LIN {X 0,Y 481.475,Z 710.731,A -85,B 0,C 180,E1 17774.011,E2 17774.011} C_VEL
LIN {X 0,Y 472.315,Z 949.794,A -85,B 0,C 180,E1 17770.464,E2 17770.464} C_VEL
LIN {X 0,Y 470.327,Z 972.285,A -85,B 0,C 180,E1 17769.967,E2 17769.967} C_VEL
LIN {X 0,Y 467.755,Z 993.239,A -85,B 0,C 180,E1 17769.33,E2 17769.33} C_VEL
LIN {X 0,Y 464.62,Z 1013.152,A -85,B 0,C 180,E1 17768.521,E2 17768.521} C_VEL
LIN {X 0,Y 460.838,Z 1033.611,A -85,B 0,C 180,E1 17767.487,E2 17767.487} C_VEL
LIN {X 0,Y 456.775,Z 1052.502,A -85,B 0,C 180,E1 17766.307,E2 17766.307} C_VEL
LIN {X 0,Y 451.974,Z 1072.368,A -85,B 0,C 180,E1 17764.802,E2 17764.802} C_VEL
LIN {X 0,Y 447.338,Z 1090.041,A -85,B 0,C 180,E1 17763.203,E2 17763.203} C_VEL
LIN {X 0,Y 442.542,Z 1106.778,A -85,B 0,C 180,E1 17761.385,E2 17761.385} C_VEL
LIN {X 0,Y 437.61,Z 1123.269,A -85,B 0,C 180,E1 17759.272,E2 17759.272} C_VEL
LIN {X 0,Y 433.368,Z 1137.028,A -85,B 0,C 180,E1 17757.182,E2 17757.182} C_VEL
LIN {X 0,Y 428.992,Z 1151.061,A -85,B 0,C 180,E1 17754.658,E2 17754.658} C_VEL
LIN {X 0,Y 425.363,Z 1163.083,A -85,B 0,C 180,E1 17752.092,E2 17752.092} C_VEL
LIN {X 0,Y 422.273,Z 1173.636,A -85,B 0,C 180,E1 17749.359,E2 17749.359} C_VEL
LIN {X 0,Y 419.714,Z 1183.269,A -85,B 0,C 180,E1 17746.326,E2 17746.326} C_VEL
LIN {X 0,Y 417.954,Z 1191.051,A -85,B 0,C 180,E1 17743.277,E2 17743.277} C_VEL
LIN {X 0,Y 416.861,Z 1196.958,A -85,B 0,C 180,E1 17740.224,E2 17740.224} C_VEL
LIN {X 0,Y 416.258,Z 1201.444,A -85,B 0,C 180,E1 17737.037,E2 17737.037} C_VEL
LIN {X 0,Y 416.044,Z 1204.09,A -85,B 0,C 180,E1 17734.134,E2 17734.134} C_VEL
LIN {X 0,Y 415.975,Z 1205.344,A -85,B 0,C 180,E1 17731.102,E2 17731.102} C_VEL
LIN {X 0,Y 415.981,Z 1205.255,A -85,B 0,C 180,E1 17728.209,E2 17728.209} C_VEL
LIN {X 0,Y 416,Z 1204.756,A -85,B 0,C 180,E1 17726.998,E2 17726.998} C_VEL
LIN {X 0,Y 415.038,Z 1204.26,A -85,B 0,C 180,E1 17725.939,E2 17725.939} C_VEL
LIN {X 0,Y 408.881,Z 1201.972,A -85,B 0,C 180,E1 17723.038,E2 17723.038} C_VEL
LIN {X 0,Y 408.362,Z 1201.086,A -85,B 0,C 180,E1 17722.189,E2 17722.189} C_VEL
LIN {X 0,Y 409.017,Z 1196.625,A -85,B 0,C 180,E1 17719.151,E2 17719.151} C_VEL
LIN {X 0,Y 410.248,Z 1190.54,A -85,B 0,C 180,E1 17716.038,E2 17716.038} C_VEL
LIN {X 0,Y 412.086,Z 1183.005,A -85,B 0,C 180,E1 17713.073,E2 17713.073} C_VEL
LIN {X 0,Y 414.825,Z 1173.243,A -85,B 0,C 180,E1 17709.985,E2 17709.985} C_VEL
LIN {X 0,Y 418.117,Z 1162.59,A -85,B 0,C 180,E1 17707.207,E2 17707.207} C_VEL
LIN {X 0,Y 421.961,Z 1150.464,A -85,B 0,C 180,E1 17704.603,E2 17704.603} C_VEL
LIN {X 0,Y 426.557,Z 1136.278,A -85,B 0,C 180,E1 17702.043,E2 17702.043} C_VEL
LIN {X 0,Y 431.32,Z 1121.527,A -85,B 0,C 180,E1 17699.799,E2 17699.799} C_VEL
LIN {X 0,Y 436.334,Z 1105.207,A -85,B 0,C 180,E1 17697.729,E2 17697.729} C_VEL
LIN {X 0,Y 441.692,Z 1086.828,A -85,B 0,C 180,E1 17695.769,E2 17695.769} C_VEL
LIN {X 0,Y 446.584,Z 1068.818,A -85,B 0,C 180,E1 17694.164,E2 17694.164} C_VEL
LIN {X 0,Y 451.18,Z 1049.908,A -85,B 0,C 180,E1 17692.772,E2 17692.772} C_VEL
LIN {X 0,Y 455.414,Z 1030.616,A -85,B 0,C 180,E1 17691.587,E2 17691.587} C_VEL
LIN {X 0,Y 459.136,Z 1010.497,A -85,B 0,C 180,E1 17690.595,E2 17690.595} C_VEL
LIN {X 0,Y 462.65,Z 987.669,A -85,B 0,C 180,E1 17689.714,E2 17689.714} C_VEL
LIN {X 0,Y 465.3,Z 965.816,A -85,B 0,C 180,E1 17689.089,E2 17689.089} C_VEL
LIN {X 0,Y 466.986,Z 943.197,A -85,B 0,C 180,E1 17688.645,E2 17688.645} C_VEL
LIN {X 0,Y 476.077,Z 710.457,A -85,B 0,C 180,E1 17685.156,E2 17685.156} C_VEL
LIN {X 0,Y 469.155,Z 656.336,A -85,B 0,C 180,E1 17683.01,E2 17683.01} C_VEL
LIN {X 0,Y 466.065,Z 634.46,A -85,B 0,C 180,E1 17682.048,E2 17682.048} C_VEL
LIN {X 0,Y 456.423,Z 617.63,A -85,B 0,C 180,E1 17680.055,E2 17680.055} C_VEL
LIN {X 0,Y 450.65,Z 602.406,A -85,B 0,C 180,E1 17677.122,E2 17677.122} C_VEL
LIN {X 0,Y 445.079,Z 588.882,A -85,B 0,C 180,E1 17674.169,E2 17674.169} C_VEL
LIN {X 0,Y 439.764,Z 577.056,A -85,B 0,C 180,E1 17671.225,E2 17671.225} C_VEL
LIN {X 0,Y 435.667,Z 568.47,A -85,B 0,C 180,E1 17668.814,E2 17668.814} C_VEL
LIN {X 0,Y 431.849,Z 560.755,A -85,B 0,C 180,E1 17666.395,E2 17666.395} C_VEL
LIN {X 0,Y 429.847,Z 556.829,A -85,B 0,C 180,E1 17665.047,E2 17665.047} C_VEL
LIN {X 0,Y 427.57,Z 552.442,A -85,B 0,C 180,E1 17663.425,E2 17663.425} C_VEL
LIN {X 0,Y 425.289,Z 548.024,A -85,B 0,C 180,E1 17661.662,E2 17661.662} C_VEL
LIN {X 0,Y 422.487,Z 542.947,A -85,B 0,C 180,E1 17659.35,E2 17659.35} C_VEL
LIN {X 0,Y 420.43,Z 539.195,A -85,B 0,C 180,E1 17657.437,E2 17657.437} C_VEL
LIN {X 0,Y 419.548,Z 537.819,A -85,B 0,C 180,E1 17656.618,E2 17656.618} C_VEL
LIN {X 0,Y 417.256,Z 533.439,A -85,B 0,C 180,E1 17653.955,E2 17653.955} C_VEL
LIN {X 0,Y 413.712,Z 527.549,A -85,B 0,C 180,E1 17648.758,E2 17648.758} C_VEL
LIN {X 0,Y 411.429,Z 524.761,A -85,B 0,C 180,E1 17643.065,E2 17643.065} C_VEL
LIN {X 0,Y 411.214,Z 524.355,A -85,B 0,C 180,E1 17639.443,E2 17639.443} C_VEL
LIN {X 0,Y 411.912,Z 525.594,A -85,B 0,C 180,E1 17635.266,E2 17635.266} C_VEL
LIN {X 0,Y 414.041,Z 528.01,A -85,B 0,C 180,E1 17631.109,E2 17631.109} C_VEL
LIN {X 0,Y 416.808,Z 532.854,A -85,B 0,C 180,E1 17626.968,E2 17626.968} C_VEL
LIN {X 0,Y 417.472,Z 534.058,A -85,B 0,C 180,E1 17626.142,E2 17626.142} C_VEL
LIN {X 0,Y 419.773,Z 538.032,A -85,B 0,C 180,E1 17623.676,E2 17623.676} C_VEL
LIN {X 0,Y 420.626,Z 539.498,A -85,B 0,C 180,E1 17622.856,E2 17622.856} C_VEL
LIN {X 0,Y 422.753,Z 543.241,A -85,B 0,C 180,E1 17620.95,E2 17620.95} C_VEL
LIN {X 0,Y 426.128,Z 549.382,A -85,B 0,C 180,E1 17618.239,E2 17618.239} C_VEL
LIN {X 0,Y 428.888,Z 554.662,A -85,B 0,C 180,E1 17616.214,E2 17616.214} C_VEL
LIN {X 0,Y 431.467,Z 559.658,A -85,B 0,C 180,E1 17614.466,E2 17614.466} C_VEL
LIN {X 0,Y 434.21,Z 565.065,A -85,B 0,C 180,E1 17612.725,E2 17612.725} C_VEL
LIN {X 0,Y 436.003,Z 567.484,A -85,B 0,C 180,E1 17612.106,E2 17612.106} C_VEL
LIN {X 0,Y 445.685,Z 579.613,A -85,B 0,C 180,E1 17609.757,E2 17609.757} C_VEL
LIN {X 0,Y 452.751,Z 588.823,A -85,B 0,C 180,E1 17608.178,E2 17608.178} C_VEL
LIN {X 0,Y 464.017,Z 604.318,A -85,B 0,C 180,E1 17605.851,E2 17605.851} C_VEL
LIN {X 0,Y 476.396,Z 623.118,A -85,B 0,C 180,E1 17603.498,E2 17603.498} C_VEL
LIN {X 0,Y 482.511,Z 633.385,A -85,B 0,C 180,E1 17602.396,E2 17602.396} C_VEL
LIN {X 0,Y 470.455,Z 868.793,A -85,B 0,C 180,E1 17598.498,E2 17598.498} C_VEL
LIN {X 0,Y 467.294,Z 928.515,A -85,B 0,C 180,E1 17597.468,E2 17597.468} C_VEL
LIN {X 0,Y 464.948,Z 952.769,A -85,B 0,C 180,E1 17596.858,E2 17596.858} C_VEL
LIN {X 0,Y 462.011,Z 976.53,A -85,B 0,C 180,E1 17596.064,E2 17596.064} C_VEL
LIN {X 0,Y 458.499,Z 999.137,A -85,B 0,C 180,E1 17595.083,E2 17595.083} C_VEL
LIN {X 0,Y 454.423,Z 1021.92,A -85,B 0,C 180,E1 17593.875,E2 17593.875} C_VEL
LIN {X 0,Y 450.215,Z 1042.26,A -85,B 0,C 180,E1 17592.568,E2 17592.568} C_VEL
LIN {X 0,Y 445.441,Z 1063.557,A -85,B 0,C 180,E1 17590.953,E2 17590.953} C_VEL
LIN {X 0,Y 440.797,Z 1082.391,A -85,B 0,C 180,E1 17589.261,E2 17589.261} C_VEL
LIN {X 0,Y 435.755,Z 1101.919,A -85,B 0,C 180,E1 17587.228,E2 17587.228} C_VEL
LIN {X 0,Y 431.061,Z 1119.183,A -85,B 0,C 180,E1 17585.116,E2 17585.116} C_VEL
LIN {X 0,Y 426.275,Z 1136.712,A -85,B 0,C 180,E1 17582.638,E2 17582.638} C_VEL
LIN {X 0,Y 422.142,Z 1151.8,A -85,B 0,C 180,E1 17580.141,E2 17580.141} C_VEL
LIN {X 0,Y 418.076,Z 1167.175,A -85,B 0,C 180,E1 17577.18,E2 17577.18} C_VEL
LIN {X 0,Y 415.095,Z 1179.144,A -85,B 0,C 180,E1 17574.475,E2 17574.475} C_VEL
LIN {X 0,Y 412.3,Z 1191.531,A -85,B 0,C 180,E1 17571.182,E2 17571.182} C_VEL
LIN {X 0,Y 410.532,Z 1200.576,A -85,B 0,C 180,E1 17568.311,E2 17568.311} C_VEL
LIN {X 0,Y 409.118,Z 1209.507,A -85,B 0,C 180,E1 17564.869,E2 17564.869} C_VEL
LIN {X 0,Y 408.428,Z 1215.42,A -85,B 0,C 180,E1 17562.01,E2 17562.01} C_VEL
LIN {X 0,Y 408.065,Z 1220.694,A -85,B 0,C 180,E1 17558.738,E2 17558.738} C_VEL
LIN {X 0,Y 407.944,Z 1223.932,A -85,B 0,C 180,E1 17555.767,E2 17555.767} C_VEL
LIN {X 0,Y 407.931,Z 1225.755,A -85,B 0,C 180,E1 17553.091,E2 17553.091} C_VEL
LIN {X 0,Y 407.957,Z 1226.572,A -85,B 0,C 180,E1 17550,E2 17550} C_VEL
LIN {X 0,Y 407.931,Z 1225.75,A -85,B 0,C 180,E1 17546.909,E2 17546.909} C_VEL
LIN {X 0,Y 407.944,Z 1223.924,A -85,B 0,C 180,E1 17544.233,E2 17544.233} C_VEL
LIN {X 0,Y 408.068,Z 1220.51,A -85,B 0,C 180,E1 17541.12,E2 17541.12} C_VEL
LIN {X 0,Y 408.428,Z 1215.403,A -85,B 0,C 180,E1 17537.99,E2 17537.99} C_VEL
LIN {X 0,Y 409.118,Z 1209.484,A -85,B 0,C 180,E1 17535.131,E2 17535.131} C_VEL
LIN {X 0,Y 410.529,Z 1200.545,A -85,B 0,C 180,E1 17531.688,E2 17531.688} C_VEL
LIN {X 0,Y 412.297,Z 1191.499,A -85,B 0,C 180,E1 17528.818,E2 17528.818} C_VEL
LIN {X 0,Y 415.091,Z 1179.102,A -85,B 0,C 180,E1 17525.524,E2 17525.524} C_VEL
LIN {X 0,Y 418.069,Z 1167.122,A -85,B 0,C 180,E1 17522.819,E2 17522.819} C_VEL
LIN {X 0,Y 421.92,Z 1152.526,A -85,B 0,C 180,E1 17519.999,E2 17519.999} C_VEL
LIN {X 0,Y 425.794,Z 1138.326,A -85,B 0,C 180,E1 17517.629,E2 17517.629} C_VEL
LIN {X 0,Y 430.766,Z 1120.127,A -85,B 0,C 180,E1 17515.018,E2 17515.018} C_VEL
LIN {X 0,Y 435.297,Z 1103.385,A -85,B 0,C 180,E1 17512.955,E2 17512.955} C_VEL
LIN {X 0,Y 440.437,Z 1083.609,A -85,B 0,C 180,E1 17510.869,E2 17510.869} C_VEL
LIN {X 0,Y 444.861,Z 1065.666,A -85,B 0,C 180,E1 17509.241,E2 17509.241} C_VEL
LIN {X 0,Y 449.965,Z 1043.149,A -85,B 0,C 180,E1 17507.506,E2 17507.506} C_VEL
LIN {X 0,Y 454.193,Z 1022.712,A -85,B 0,C 180,E1 17506.185,E2 17506.185} C_VEL
LIN {X 0,Y 458.357,Z 999.55,A -85,B 0,C 180,E1 17504.948,E2 17504.948} C_VEL
LIN {X 0,Y 461.835,Z 977.187,A -85,B 0,C 180,E1 17503.974,E2 17503.974} C_VEL
LIN {X 0,Y 464.833,Z 953.099,A -85,B 0,C 180,E1 17503.163,E2 17503.163} C_VEL
LIN {X 0,Y 467.187,Z 928.855,A -85,B 0,C 180,E1 17502.549,E2 17502.549} C_VEL
LIN {X 0,Y 470.286,Z 870.553,A -85,B 0,C 180,E1 17501.542,E2 17501.542} C_VEL
LIN {X 0,Y 482.429,Z 633.121,A -85,B 0,C 180,E1 17497.61,E2 17497.61} C_VEL
LIN {X 0,Y 471.756,Z 615.97,A -85,B 0,C 180,E1 17495.671,E2 17495.671} C_VEL
LIN {X 0,Y 460.86,Z 599.95,A -85,B 0,C 180,E1 17493.553,E2 17493.553} C_VEL
LIN {X 0,Y 450.245,Z 585.446,A -85,B 0,C 180,E1 17491.31,E2 17491.31} C_VEL
LIN {X 0,Y 442.161,Z 575.196,A -85,B 0,C 180,E1 17489.462,E2 17489.462} C_VEL
LIN {X 0,Y 434.621,Z 565.798,A -85,B 0,C 180,E1 17487.544,E2 17487.544} C_VEL
LIN {X 0,Y 430.622,Z 557.777,A -85,B 0,C 180,E1 17484.999,E2 17484.999} C_VEL
LIN {X 0,Y 427.83,Z 552.655,A -85,B 0,C 180,E1 17483.119,E2 17483.119} C_VEL
LIN {X 0,Y 425.283,Z 547.918,A -85,B 0,C 180,E1 17481.228,E2 17481.228} C_VEL
LIN {X 0,Y 423.196,Z 543.745,A -85,B 0,C 180,E1 17479.46,E2 17479.46} C_VEL
LIN {X 0,Y 420.729,Z 539.878,A -85,B 0,C 180,E1 17477.425,E2 17477.425} C_VEL
LIN {X 0,Y 419.952,Z 538.228,A -85,B 0,C 180,E1 17476.602,E2 17476.602} C_VEL
LIN {X 0,Y 417.45,Z 534.026,A -85,B 0,C 180,E1 17474,E2 17474} C_VEL
LIN {X 0,Y 416.779,Z 532.794,A -85,B 0,C 180,E1 17473.174,E2 17473.174} C_VEL
LIN {X 0,Y 414.104,Z 528.173,A -85,B 0,C 180,E1 17469.31,E2 17469.31} C_VEL
LIN {X 0,Y 411.835,Z 525.452,A -85,B 0,C 180,E1 17465.014,E2 17465.014} C_VEL
LIN {X 0,Y 411.092,Z 524.019,A -85,B 0,C 180,E1 17460.836,E2 17460.836} C_VEL
LIN {X 0,Y 411.206,Z 524.285,A -85,B 0,C 180,E1 17457.352,E2 17457.352} C_VEL
LIN {X 0,Y 412.766,Z 526.643,A -85,B 0,C 180,E1 17452.343,E2 17452.343} C_VEL
LIN {X 0,Y 414.092,Z 528.295,A -85,B 0,C 180,E1 17450.112,E2 17450.112} C_VEL
LIN {X 0,Y 417.371,Z 533.826,A -85,B 0,C 180,E1 17445.573,E2 17445.573} C_VEL
LIN {X 0,Y 419.445,Z 537.704,A -85,B 0,C 180,E1 17443.235,E2 17443.235} C_VEL
LIN {X 0,Y 420.365,Z 539.033,A -85,B 0,C 180,E1 17442.417,E2 17442.417} C_VEL
LIN {X 0,Y 422.698,Z 543.207,A -85,B 0,C 180,E1 17440.294,E2 17440.294} C_VEL
LIN {X 0,Y 426.088,Z 549.604,A -85,B 0,C 180,E1 17437.511,E2 17437.511} C_VEL
LIN {X 0,Y 428.664,Z 554.517,A -85,B 0,C 180,E1 17435.615,E2 17435.615} C_VEL
LIN {X 0,Y 431.329,Z 559.755,A -85,B 0,C 180,E1 17433.779,E2 17433.779} C_VEL
LIN {X 0,Y 435.167,Z 567.3,A -85,B 0,C 180,E1 17431.366,E2 17431.366} C_VEL
LIN {X 0,Y 440.752,Z 579.074,A -85,B 0,C 180,E1 17428.09,E2 17428.09} C_VEL
LIN {X 0,Y 446.612,Z 592.479,A -85,B 0,C 180,E1 17424.873,E2 17424.873} C_VEL
LIN {X 0,Y 452.53,Z 607.236,A -85,B 0,C 180,E1 17421.78,E2 17421.78} C_VEL
LIN {X 0,Y 456.803,Z 618.552,A -85,B 0,C 180,E1 17419.698,E2 17419.698} C_VEL
LIN {X 0,Y 466.093,Z 634.647,A -85,B 0,C 180,E1 17417.819,E2 17417.819} C_VEL
LIN {X 0,Y 472.808,Z 685.178,A -85,B 0,C 180,E1 17415.711,E2 17415.711} C_VEL
LIN {X 0,Y 476.03,Z 712.189,A -85,B 0,C 180,E1 17414.7,E2 17414.7} C_VEL
LIN {X 0,Y 466.553,Z 949.506,A -85,B 0,C 180,E1 17411.147,E2 17411.147} C_VEL
LIN {X 0,Y 464.513,Z 972,A -85,B 0,C 180,E1 17410.647,E2 17410.647} C_VEL
LIN {X 0,Y 461.762,Z 993.624,A -85,B 0,C 180,E1 17409.983,E2 17409.983} C_VEL
LIN {X 0,Y 458.53,Z 1013.516,A -85,B 0,C 180,E1 17409.166,E2 17409.166} C_VEL
LIN {X 0,Y 454.319,Z 1035.316,A -85,B 0,C 180,E1 17408.04,E2 17408.04} C_VEL
LIN {X 0,Y 450.162,Z 1054.016,A -85,B 0,C 180,E1 17406.848,E2 17406.848} C_VEL
LIN {X 0,Y 445.418,Z 1072.868,A -85,B 0,C 180,E1 17405.391,E2 17405.391} C_VEL
LIN {X 0,Y 440.636,Z 1090.48,A -85,B 0,C 180,E1 17403.775,E2 17403.775} C_VEL
LIN {X 0,Y 435.686,Z 1107.158,A -85,B 0,C 180,E1 17401.936,E2 17401.936} C_VEL
LIN {X 0,Y 430.583,Z 1123.597,A -85,B 0,C 180,E1 17399.797,E2 17399.797} C_VEL
LIN {X 0,Y 425.932,Z 1138.158,A -85,B 0,C 180,E1 17397.545,E2 17397.545} C_VEL
LIN {X 0,Y 421.639,Z 1151.337,A -85,B 0,C 180,E1 17395.117,E2 17395.117} C_VEL
LIN {X 0,Y 417.856,Z 1163.336,A -85,B 0,C 180,E1 17392.51,E2 17392.51} C_VEL
LIN {X 0,Y 414.624,Z 1173.88,A -85,B 0,C 180,E1 17389.731,E2 17389.731} C_VEL
LIN {X 0,Y 411.937,Z 1183.499,A -85,B 0,C 180,E1 17386.643,E2 17386.643} C_VEL
LIN {X 0,Y 410.153,Z 1190.967,A -85,B 0,C 180,E1 17383.678,E2 17383.678} C_VEL
LIN {X 0,Y 408.96,Z 1196.931,A -85,B 0,C 180,E1 17380.566,E2 17380.566} C_VEL
LIN {X 0,Y 408.299,Z 1201.502,A -85,B 0,C 180,E1 17377.316,E2 17377.316} C_VEL
LIN {X 0,Y 408.057,Z 1204.189,A -85,B 0,C 180,E1 17374.356,E2 17374.356} C_VEL
LIN {X 0,Y 407.977,Z 1205.549,A -85,B 0,C 180,E1 17371.123,E2 17371.123} C_VEL
LIN {X 0,Y 407.985,Z 1205.459,A -85,B 0,C 180,E1 17368.174,E2 17368.174} C_VEL
LIN {X 0,Y 408.077,Z 1203.842,A -85,B 0,C 180,E1 17365.081,E2 17365.081} C_VEL
LIN {X 0,Y 408.362,Z 1201.086,A -85,B 0,C 180,E1 17362.189,E2 17362.189} C_VEL
LIN {X 0,Y 407.563,Z 1199.87,A -85,B 0,C 180,E1 17361.118,E2 17361.118} C_VEL
LIN {X 0,Y 401.991,Z 1195.591,A -85,B 0,C 180,E1 17358.19,E2 17358.19} C_VEL
LIN {X 0,Y 401.659,Z 1194.002,A -85,B 0,C 180,E1 17357.347,E2 17357.347} C_VEL
LIN {X 0,Y 403.325,Z 1187.057,A -85,B 0,C 180,E1 17354.175,E2 17354.175} C_VEL
LIN {X 0,Y 405.654,Z 1178.602,A -85,B 0,C 180,E1 17351.162,E2 17351.162} C_VEL
LIN {X 0,Y 408.82,Z 1168.389,A -85,B 0,C 180,E1 17348.177,E2 17348.177} C_VEL
LIN {X 0,Y 412.449,Z 1157.336,A -85,B 0,C 180,E1 17345.51,E2 17345.51} C_VEL
LIN {X 0,Y 416.86,Z 1144.169,A -85,B 0,C 180,E1 17342.86,E2 17342.86} C_VEL
LIN {X 0,Y 421.678,Z 1129.954,A -85,B 0,C 180,E1 17340.449,E2 17340.449} C_VEL
LIN {X 0,Y 426.626,Z 1114.752,A -85,B 0,C 180,E1 17338.296,E2 17338.296} C_VEL
LIN {X 0,Y 432.16,Z 1097.081,A -85,B 0,C 180,E1 17336.191,E2 17336.191} C_VEL
LIN {X 0,Y 437.37,Z 1079.399,A -85,B 0,C 180,E1 17334.423,E2 17334.423} C_VEL
LIN {X 0,Y 442.34,Z 1060.665,A -85,B 0,C 180,E1 17332.878,E2 17332.878} C_VEL
LIN {X 0,Y 447.267,Z 1040.04,A -85,B 0,C 180,E1 17331.468,E2 17331.468} C_VEL
LIN {X 0,Y 451.429,Z 1020.168,A -85,B 0,C 180,E1 17330.366,E2 17330.366} C_VEL
LIN {X 0,Y 454.999,Z 999.732,A -85,B 0,C 180,E1 17329.465,E2 17329.465} C_VEL
LIN {X 0,Y 458.124,Z 978.166,A -85,B 0,C 180,E1 17328.726,E2 17328.726} C_VEL
LIN {X 0,Y 460.408,Z 956.246,A -85,B 0,C 180,E1 17328.192,E2 17328.192} C_VEL
LIN {X 0,Y 462.012,Z 926.812,A -85,B 0,C 180,E1 17327.692,E2 17327.692} C_VEL
LIN {X 0,Y 470.705,Z 711.851,A -85,B 0,C 180,E1 17324.447,E2 17324.447} C_VEL
LIN {X 0,Y 463.893,Z 656.921,A -85,B 0,C 180,E1 17322.229,E2 17322.229} C_VEL
LIN {X 0,Y 461.328,Z 638.734,A -85,B 0,C 180,E1 17321.404,E2 17321.404} C_VEL
LIN {X 0,Y 451.533,Z 621.923,A -85,B 0,C 180,E1 17319.358,E2 17319.358} C_VEL
LIN {X 0,Y 448.032,Z 615.791,A -85,B 0,C 180,E1 17318.511,E2 17318.511} C_VEL
LIN {X 0,Y 442.416,Z 601.276,A -85,B 0,C 180,E1 17315.51,E2 17315.51} C_VEL
LIN {X 0,Y 437.07,Z 588.547,A -85,B 0,C 180,E1 17312.521,E2 17312.521} C_VEL
LIN {X 0,Y 431.58,Z 576.489,A -85,B 0,C 180,E1 17309.265,E2 17309.265} C_VEL
LIN {X 0,Y 426.758,Z 566.737,A -85,B 0,C 180,E1 17306.19,E2 17306.19} C_VEL
LIN {X 0,Y 424.709,Z 562.697,A -85,B 0,C 180,E1 17304.776,E2 17304.776} C_VEL
LIN {X 0,Y 422.672,Z 558.665,A -85,B 0,C 180,E1 17303.27,E2 17303.27} C_VEL
LIN {X 0,Y 420.217,Z 554.001,A -85,B 0,C 180,E1 17301.35,E2 17301.35} C_VEL
LIN {X 0,Y 417.845,Z 549.444,A -85,B 0,C 180,E1 17299.283,E2 17299.283} C_VEL
LIN {X 0,Y 415.686,Z 545.419,A -85,B 0,C 180,E1 17297.209,E2 17297.209} C_VEL
LIN {X 0,Y 412.707,Z 540.045,A -85,B 0,C 180,E1 17293.878,E2 17293.878} C_VEL
LIN {X 0,Y 409.293,Z 534.215,A -85,B 0,C 180,E1 17288.712,E2 17288.712} C_VEL
LIN {X 0,Y 407.081,Z 531.49,A -85,B 0,C 180,E1 17283.098,E2 17283.098} C_VEL
LIN {X 0,Y 406.871,Z 531.074,A -85,B 0,C 180,E1 17279.437,E2 17279.437} C_VEL
LIN {X 0,Y 407.533,Z 532.273,A -85,B 0,C 180,E1 17275.356,E2 17275.356} C_VEL
LIN {X 0,Y 409.63,Z 534.694,A -85,B 0,C 180,E1 17271.154,E2 17271.154} C_VEL
LIN {X 0,Y 412.396,Z 539.532,A -85,B 0,C 180,E1 17266.968,E2 17266.968} C_VEL
LIN {X 0,Y 415.53,Z 544.915,A -85,B 0,C 180,E1 17263.504,E2 17263.504} C_VEL
LIN {X 0,Y 417.938,Z 549.544,A -85,B 0,C 180,E1 17261.157,E2 17261.157} C_VEL
LIN {X 0,Y 418.733,Z 550.985,A -85,B 0,C 180,E1 17260.47,E2 17260.47} C_VEL
LIN {X 0,Y 421.283,Z 555.629,A -85,B 0,C 180,E1 17258.415,E2 17258.415} C_VEL
LIN {X 0,Y 423.996,Z 560.913,A -85,B 0,C 180,E1 17256.365,E2 17256.365} C_VEL
LIN {X 0,Y 426.536,Z 565.917,A -85,B 0,C 180,E1 17254.596,E2 17254.596} C_VEL
LIN {X 0,Y 428.064,Z 568.339,A -85,B 0,C 180,E1 17253.876,E2 17253.876} C_VEL
LIN {X 0,Y 437.634,Z 579.911,A -85,B 0,C 180,E1 17251.365,E2 17251.365} C_VEL
LIN {X 0,Y 448.111,Z 593.353,A -85,B 0,C 180,E1 17248.898,E2 17248.898} C_VEL
LIN {X 0,Y 460.717,Z 611.066,A -85,B 0,C 180,E1 17246.211,E2 17246.211} C_VEL
LIN {X 0,Y 472.675,Z 629.484,A -85,B 0,C 180,E1 17243.885,E2 17243.885} C_VEL
LIN {X 0,Y 477.105,Z 636.908,A -85,B 0,C 180,E1 17243.066,E2 17243.066} C_VEL
LIN {X 0,Y 464.688,Z 872.136,A -85,B 0,C 180,E1 17239.145,E2 17239.145} C_VEL
LIN {X 0,Y 461.581,Z 928.938,A -85,B 0,C 180,E1 17238.157,E2 17238.157} C_VEL
LIN {X 0,Y 459.173,Z 953.102,A -85,B 0,C 180,E1 17237.544,E2 17237.544} C_VEL
LIN {X 0,Y 456.14,Z 976.899,A -85,B 0,C 180,E1 17236.743,E2 17236.743} C_VEL
LIN {X 0,Y 452.544,Z 999.372,A -85,B 0,C 180,E1 17235.761,E2 17235.761} C_VEL
LIN {X 0,Y 448.263,Z 1022.504,A -85,B 0,C 180,E1 17234.522,E2 17234.522} C_VEL
LIN {X 0,Y 443.942,Z 1042.708,A -85,B 0,C 180,E1 17233.21,E2 17233.21} C_VEL
LIN {X 0,Y 438.856,Z 1064.54,A -85,B 0,C 180,E1 17231.528,E2 17231.528} C_VEL
LIN {X 0,Y 434.069,Z 1083.282,A -85,B 0,C 180,E1 17229.819,E2 17229.819} C_VEL
LIN {X 0,Y 428.637,Z 1103.417,A -85,B 0,C 180,E1 17227.673,E2 17227.673} C_VEL
LIN {X 0,Y 424.004,Z 1119.851,A -85,B 0,C 180,E1 17225.624,E2 17225.624} C_VEL
LIN {X 0,Y 418.797,Z 1138.077,A -85,B 0,C 180,E1 17222.979,E2 17222.979} C_VEL
LIN {X 0,Y 414.75,Z 1152.284,A -85,B 0,C 180,E1 17220.575,E2 17220.575} C_VEL
LIN {X 0,Y 410.488,Z 1167.653,A -85,B 0,C 180,E1 17217.544,E2 17217.544} C_VEL
LIN {X 0,Y 407.335,Z 1179.788,A -85,B 0,C 180,E1 17214.736,E2 17214.736} C_VEL
LIN {X 0,Y 404.492,Z 1191.761,A -85,B 0,C 180,E1 17211.459,E2 17211.459} C_VEL
LIN {X 0,Y 402.644,Z 1200.759,A -85,B 0,C 180,E1 17208.533,E2 17208.533} C_VEL
LIN {X 0,Y 401.165,Z 1209.599,A -85,B 0,C 180,E1 17205.023,E2 17205.023} C_VEL
LIN {X 0,Y 400.445,Z 1215.468,A -85,B 0,C 180,E1 17202.107,E2 17202.107} C_VEL
LIN {X 0,Y 400.059,Z 1220.823,A -85,B 0,C 180,E1 17198.624,E2 17198.624} C_VEL
LIN {X 0,Y 399.943,Z 1223.869,A -85,B 0,C 180,E1 17195.71,E2 17195.71} C_VEL
LIN {X 0,Y 399.93,Z 1225.694,A -85,B 0,C 180,E1 17192.866,E2 17192.866} C_VEL
LIN {X 0,Y 399.944,Z 1226.326,A -85,B 0,C 180,E1 17189.714,E2 17189.714} C_VEL
LIN {X 0,Y 399.933,Z 1225.544,A -85,B 0,C 180,E1 17186.847,E2 17186.847} C_VEL
LIN {X 0,Y 399.951,Z 1223.716,A -85,B 0,C 180,E1 17184.117,E2 17184.117} C_VEL
LIN {X 0,Y 400.077,Z 1220.296,A -85,B 0,C 180,E1 17180.941,E2 17180.941} C_VEL
LIN {X 0,Y 400.474,Z 1215.182,A -85,B 0,C 180,E1 17177.748,E2 17177.748} C_VEL
LIN {X 0,Y 401.213,Z 1209.256,A -85,B 0,C 180,E1 17174.831,E2 17174.831} C_VEL
LIN {X 0,Y 402.718,Z 1200.302,A -85,B 0,C 180,E1 17171.32,E2 17171.32} C_VEL
LIN {X 0,Y 404.601,Z 1191.247,A -85,B 0,C 180,E1 17168.395,E2 17168.395} C_VEL
LIN {X 0,Y 407.555,Z 1178.828,A -85,B 0,C 180,E1 17165.041,E2 17165.041} C_VEL
LIN {X 0,Y 410.692,Z 1166.837,A -85,B 0,C 180,E1 17162.29,E2 17162.29} C_VEL
LIN {X 0,Y 414.813,Z 1151.945,A -85,B 0,C 180,E1 17159.377,E2 17159.377} C_VEL
LIN {X 0,Y 419.039,Z 1137.118,A -85,B 0,C 180,E1 17156.879,E2 17156.879} C_VEL
LIN {X 0,Y 423.993,Z 1119.745,A -85,B 0,C 180,E1 17154.375,E2 17154.375} C_VEL
LIN {X 0,Y 428.622,Z 1103.294,A -85,B 0,C 180,E1 17152.326,E2 17152.326} C_VEL
LIN {X 0,Y 433.925,Z 1083.609,A -85,B 0,C 180,E1 17150.227,E2 17150.227} C_VEL
LIN {X 0,Y 438.645,Z 1065.112,A -85,B 0,C 180,E1 17148.534,E2 17148.534} C_VEL
LIN {X 0,Y 443.722,Z 1043.41,A -85,B 0,C 180,E1 17146.852,E2 17146.852} C_VEL
LIN {X 0,Y 448.086,Z 1022.997,A -85,B 0,C 180,E1 17145.52,E2 17145.52} C_VEL
LIN {X 0,Y 452.402,Z 999.751,A -85,B 0,C 180,E1 17144.269,E2 17144.269} C_VEL
LIN {X 0,Y 455.884,Z 978.019,A -85,B 0,C 180,E1 17143.314,E2 17143.314} C_VEL
LIN {X 0,Y 459.022,Z 953.699,A -85,B 0,C 180,E1 17142.485,E2 17142.485} C_VEL
LIN {X 0,Y 461.444,Z 929.538,A -85,B 0,C 180,E1 17141.867,E2 17141.867} C_VEL
LIN {X 0,Y 464.355,Z 877.024,A -85,B 0,C 180,E1 17140.948,E2 17140.948} C_VEL
LIN {X 0,Y 476.844,Z 639.834,A -85,B 0,C 180,E1 17136.992,E2 17136.992} C_VEL
LIN {X 0,Y 476.901,Z 636.451,A -85,B 0,C 180,E1 17136.919,E2 17136.919} C_VEL
LIN {X 0,Y 465.03,Z 617.552,A -85,B 0,C 180,E1 17134.68,E2 17134.68} C_VEL
LIN {X 0,Y 453.999,Z 601.561,A -85,B 0,C 180,E1 17132.431,E2 17132.431} C_VEL
LIN {X 0,Y 443.916,Z 587.959,A -85,B 0,C 180,E1 17130.189,E2 17130.189} C_VEL
LIN {X 0,Y 435.274,Z 577.072,A -85,B 0,C 180,E1 17128.094,E2 17128.094} C_VEL
LIN {X 0,Y 427.323,Z 567.417,A -85,B 0,C 180,E1 17125.948,E2 17125.948} C_VEL
LIN {X 0,Y 424.971,Z 562.912,A -85,B 0,C 180,E1 17124.423,E2 17124.423} C_VEL
LIN {X 0,Y 422.957,Z 558.896,A -85,B 0,C 180,E1 17122.959,E2 17122.959} C_VEL
LIN {X 0,Y 420.437,Z 554.175,A -85,B 0,C 180,E1 17121.046,E2 17121.046} C_VEL
LIN {X 0,Y 417.986,Z 549.59,A -85,B 0,C 180,E1 17118.986,E2 17118.986} C_VEL
LIN {X 0,Y 415.899,Z 545.786,A -85,B 0,C 180,E1 17117.056,E2 17117.056} C_VEL
LIN {X 0,Y 412.746,Z 539.998,A -85,B 0,C 180,E1 17113.591,E2 17113.591} C_VEL
LIN {X 0,Y 409.29,Z 534.222,A -85,B 0,C 180,E1 17108.57,E2 17108.57} C_VEL
LIN {X 0,Y 406.954,Z 531.219,A -85,B 0,C 180,E1 17102.817,E2 17102.817} C_VEL
LIN {X 0,Y 406.741,Z 530.682,A -85,B 0,C 180,E1 17099.014,E2 17099.014} C_VEL
LIN {X 0,Y 407.38,Z 532,A -85,B 0,C 180,E1 17094.789,E2 17094.789} C_VEL
LIN {X 0,Y 409.598,Z 534.78,A -85,B 0,C 180,E1 17090.303,E2 17090.303} C_VEL
LIN {X 0,Y 412.354,Z 539.517,A -85,B 0,C 180,E1 17086.253,E2 17086.253} C_VEL
LIN {X 0,Y 415.174,Z 544.569,A -85,B 0,C 180,E1 17083.057,E2 17083.057} C_VEL
LIN {X 0,Y 418.539,Z 550.807,A -85,B 0,C 180,E1 17079.878,E2 17079.878} C_VEL
LIN {X 0,Y 421.207,Z 555.834,A -85,B 0,C 180,E1 17077.677,E2 17077.677} C_VEL
LIN {X 0,Y 423.739,Z 560.755,A -85,B 0,C 180,E1 17075.758,E2 17075.758} C_VEL
LIN {X 0,Y 426.45,Z 566.166,A -85,B 0,C 180,E1 17073.845,E2 17073.845} C_VEL
LIN {X 0,Y 430.072,Z 573.457,A -85,B 0,C 180,E1 17071.497,E2 17071.497} C_VEL
LIN {X 0,Y 435.199,Z 584.385,A -85,B 0,C 180,E1 17068.41,E2 17068.41} C_VEL
LIN {X 0,Y 440.958,Z 597.738,A -85,B 0,C 180,E1 17065.15,E2 17065.15} C_VEL
LIN {X 0,Y 446.775,Z 612.484,A -85,B 0,C 180,E1 17062.015,E2 17062.015} C_VEL
LIN {X 0,Y 448.784,Z 617.439,A -85,B 0,C 180,E1 17061.116,E2 17061.116} C_VEL
LIN {X 0,Y 458.841,Z 634.549,A -85,B 0,C 180,E1 17058.968,E2 17058.968} C_VEL
LIN {X 0,Y 461.445,Z 639.373,A -85,B 0,C 180,E1 17058.435,E2 17058.435} C_VEL
LIN {X 0,Y 467.889,Z 689.514,A -85,B 0,C 180,E1 17056.317,E2 17056.317} C_VEL
LIN {X 0,Y 470.653,Z 713.641,A -85,B 0,C 180,E1 17055.404,E2 17055.404} C_VEL
LIN {X 0,Y 460.859,Z 949.204,A -85,B 0,C 180,E1 17051.846,E2 17051.846} C_VEL
LIN {X 0,Y 458.751,Z 971.837,A -85,B 0,C 180,E1 17051.34,E2 17051.34} C_VEL
LIN {X 0,Y 455.951,Z 993.257,A -85,B 0,C 180,E1 17050.68,E2 17050.68} C_VEL
LIN {X 0,Y 452.561,Z 1013.526,A -85,B 0,C 180,E1 17049.844,E2 17049.844} C_VEL
LIN {X 0,Y 448.295,Z 1035.024,A -85,B 0,C 180,E1 17048.727,E2 17048.727} C_VEL
LIN {X 0,Y 444.004,Z 1053.747,A -85,B 0,C 180,E1 17047.527,E2 17047.527} C_VEL
LIN {X 0,Y 439.14,Z 1072.521,A -85,B 0,C 180,E1 17046.068,E2 17046.068} C_VEL
LIN {X 0,Y 433.977,Z 1090.896,A -85,B 0,C 180,E1 17044.365,E2 17044.365} C_VEL
LIN {X 0,Y 428.873,Z 1107.537,A -85,B 0,C 180,E1 17042.505,E2 17042.505} C_VEL
LIN {X 0,Y 423.289,Z 1124.823,A -85,B 0,C 180,E1 17040.207,E2 17040.207} C_VEL
LIN {X 0,Y 418.322,Z 1139.844,A -85,B 0,C 180,E1 17037.823,E2 17037.823} C_VEL
LIN {X 0,Y 413.861,Z 1152.968,A -85,B 0,C 180,E1 17035.316,E2 17035.316} C_VEL
LIN {X 0,Y 409.622,Z 1165.794,A -85,B 0,C 180,E1 17032.382,E2 17032.382} C_VEL
LIN {X 0,Y 406.423,Z 1176.09,A -85,B 0,C 180,E1 17029.547,E2 17029.547} C_VEL
LIN {X 0,Y 403.862,Z 1184.889,A -85,B 0,C 180,E1 17026.541,E2 17026.541} C_VEL
LIN {X 0,Y 401.939,Z 1192.639,A -85,B 0,C 180,E1 17023.23,E2 17023.23} C_VEL
LIN {X 0,Y 400.839,Z 1198.352,A -85,B 0,C 180,E1 17020.056,E2 17020.056} C_VEL
LIN {X 0,Y 400.253,Z 1202.313,A -85,B 0,C 180,E1 17016.887,E2 17016.887} C_VEL
LIN {X 0,Y 400.026,Z 1204.914,A -85,B 0,C 180,E1 17013.583,E2 17013.583} C_VEL
LIN {X 0,Y 399.981,Z 1205.817,A -85,B 0,C 180,E1 17010.716,E2 17010.716} C_VEL
LIN {X 0,Y 399.999,Z 1205.408,A -85,B 0,C 180,E1 17007.421,E2 17007.421} C_VEL
LIN {X 0,Y 400.126,Z 1203.62,A -85,B 0,C 180,E1 17004.407,E2 17004.407} C_VEL
LIN {X 0,Y 400.552,Z 1200.071,A -85,B 0,C 180,E1 17001.097,E2 17001.097} C_VEL
LIN {X 0,Y 401.442,Z 1195.146,A -85,B 0,C 180,E1 16997.924,E2 16997.924} C_VEL
LIN {X 0,Y 401.659,Z 1194.002,A -85,B 0,C 180,E1 16997.347,E2 16997.347} C_VEL
LIN {X 0,Y 401.125,Z 1191.983,A -85,B 0,C 180,E1 16996.282,E2 16996.282} C_VEL
LIN {X 0,Y 396.563,Z 1186.1,A -85,B 0,C 180,E1 16993.42,E2 16993.42} C_VEL
LIN {X 0,Y 396.495,Z 1183.78,A -85,B 0,C 180,E1 16992.513,E2 16992.513} C_VEL
LIN {X 0,Y 399.606,Z 1173.721,A -85,B 0,C 180,E1 16989.188,E2 16989.188} C_VEL
LIN {X 0,Y 403.197,Z 1163.104,A -85,B 0,C 180,E1 16986.314,E2 16986.314} C_VEL
LIN {X 0,Y 407.378,Z 1150.986,A -85,B 0,C 180,E1 16983.622,E2 16983.622} C_VEL
LIN {X 0,Y 412.328,Z 1136.878,A -85,B 0,C 180,E1 16980.989,E2 16980.989} C_VEL
LIN {X 0,Y 417.437,Z 1122.161,A -85,B 0,C 180,E1 16978.684,E2 16978.684} C_VEL
LIN {X 0,Y 422.796,Z 1105.943,A -85,B 0,C 180,E1 16976.563,E2 16976.563} C_VEL
LIN {X 0,Y 428.317,Z 1088.361,A -85,B 0,C 180,E1 16974.625,E2 16974.625} C_VEL
LIN {X 0,Y 433.277,Z 1071.229,A -85,B 0,C 180,E1 16973.048,E2 16973.048} C_VEL
LIN {X 0,Y 438.566,Z 1051.117,A -85,B 0,C 180,E1 16971.509,E2 16971.509} C_VEL
LIN {X 0,Y 443.267,Z 1031.06,A -85,B 0,C 180,E1 16970.247,E2 16970.247} C_VEL
LIN {X 0,Y 447.201,Z 1011.056,A -85,B 0,C 180,E1 16969.243,E2 16969.243} C_VEL
LIN {X 0,Y 450.823,Z 989.276,A -85,B 0,C 180,E1 16968.377,E2 16968.377} C_VEL
LIN {X 0,Y 453.553,Z 968.284,A -85,B 0,C 180,E1 16967.756,E2 16967.756} C_VEL
LIN {X 0,Y 455.55,Z 945.17,A -85,B 0,C 180,E1 16967.27,E2 16967.27} C_VEL
LIN {X 0,Y 465.42,Z 713.372,A -85,B 0,C 180,E1 16963.728,E2 16963.728} C_VEL
LIN {X 0,Y 458.863,Z 658.818,A -85,B 0,C 180,E1 16961.486,E2 16961.486} C_VEL
LIN {X 0,Y 456.822,Z 643.395,A -85,B 0,C 180,E1 16960.787,E2 16960.787} C_VEL
LIN {X 0,Y 446.974,Z 626.414,A -85,B 0,C 180,E1 16958.66,E2 16958.66} C_VEL
LIN {X 0,Y 439.738,Z 614.194,A -85,B 0,C 180,E1 16956.891,E2 16956.891} C_VEL
LIN {X 0,Y 434.154,Z 600.139,A -85,B 0,C 180,E1 16953.759,E2 16953.759} C_VEL
LIN {X 0,Y 428.891,Z 588.024,A -85,B 0,C 180,E1 16950.657,E2 16950.657} C_VEL
LIN {X 0,Y 424.428,Z 578.225,A -85,B 0,C 180,E1 16947.805,E2 16947.805} C_VEL
LIN {X 0,Y 419.994,Z 569.27,A -85,B 0,C 180,E1 16944.772,E2 16944.772} C_VEL
LIN {X 0,Y 417.576,Z 564.575,A -85,B 0,C 180,E1 16942.974,E2 16942.974} C_VEL
LIN {X 0,Y 415.552,Z 560.508,A -85,B 0,C 180,E1 16941.305,E2 16941.305} C_VEL
LIN {X 0,Y 413.016,Z 555.718,A -85,B 0,C 180,E1 16939.076,E2 16939.076} C_VEL
LIN {X 0,Y 410.491,Z 551.004,A -85,B 0,C 180,E1 16936.559,E2 16936.559} C_VEL
LIN {X 0,Y 408.208,Z 546.811,A -85,B 0,C 180,E1 16933.889,E2 16933.889} C_VEL
LIN {X 0,Y 404.876,Z 540.881,A -85,B 0,C 180,E1 16928.664,E2 16928.664} C_VEL
LIN {X 0,Y 402.715,Z 538.17,A -85,B 0,C 180,E1 16922.989,E2 16922.989} C_VEL
LIN {X 0,Y 402.529,Z 537.793,A -85,B 0,C 180,E1 16919.431,E2 16919.431} C_VEL
LIN {X 0,Y 403.2,Z 539.011,A -85,B 0,C 180,E1 16915.306,E2 16915.306} C_VEL
LIN {X 0,Y 405.216,Z 541.381,A -85,B 0,C 180,E1 16911.2,E2 16911.2} C_VEL
LIN {X 0,Y 407.979,Z 546.206,A -85,B 0,C 180,E1 16906.969,E2 16906.969} C_VEL
LIN {X 0,Y 410.766,Z 551.252,A -85,B 0,C 180,E1 16903.744,E2 16903.744} C_VEL
LIN {X 0,Y 413.523,Z 556.268,A -85,B 0,C 180,E1 16901.094,E2 16901.094} C_VEL
LIN {X 0,Y 416.578,Z 562.262,A -85,B 0,C 180,E1 16898.455,E2 16898.455} C_VEL
LIN {X 0,Y 419.105,Z 567.159,A -85,B 0,C 180,E1 16896.52,E2 16896.52} C_VEL
LIN {X 0,Y 420.6,Z 569.698,A -85,B 0,C 180,E1 16895.678,E2 16895.678} C_VEL
LIN {X 0,Y 430.676,Z 581.619,A -85,B 0,C 180,E1 16892.82,E2 16892.82} C_VEL
LIN {X 0,Y 440.132,Z 593.765,A -85,B 0,C 180,E1 16890.426,E2 16890.426} C_VEL
LIN {X 0,Y 449.165,Z 605.93,A -85,B 0,C 180,E1 16888.345,E2 16888.345} C_VEL
LIN {X 0,Y 460.237,Z 621.989,A -85,B 0,C 180,E1 16886.002,E2 16886.002} C_VEL
LIN {X 0,Y 471.759,Z 640.423,A -85,B 0,C 180,E1 16883.752,E2 16883.752} C_VEL
LIN {X 0,Y 459.106,Z 873.265,A -85,B 0,C 180,E1 16879.846,E2 16879.846} C_VEL
LIN {X 0,Y 455.932,Z 929.409,A -85,B 0,C 180,E1 16878.862,E2 16878.862} C_VEL
LIN {X 0,Y 453.448,Z 953.603,A -85,B 0,C 180,E1 16878.243,E2 16878.243} C_VEL
LIN {X 0,Y 450.263,Z 977.724,A -85,B 0,C 180,E1 16877.421,E2 16877.421} C_VEL
LIN {X 0,Y 446.617,Z 999.834,A -85,B 0,C 180,E1 16876.447,E2 16876.447} C_VEL
LIN {X 0,Y 442.065,Z 1023.538,A -85,B 0,C 180,E1 16875.159,E2 16875.159} C_VEL
LIN {X 0,Y 437.563,Z 1043.903,A -85,B 0,C 180,E1 16873.818,E2 16873.818} C_VEL
LIN {X 0,Y 432.121,Z 1066.276,A -85,B 0,C 180,E1 16872.056,E2 16872.056} C_VEL
LIN {X 0,Y 427.383,Z 1084.177,A -85,B 0,C 180,E1 16870.394,E2 16870.394} C_VEL
LIN {X 0,Y 421.683,Z 1104.456,A -85,B 0,C 180,E1 16868.188,E2 16868.188} C_VEL
LIN {X 0,Y 416.767,Z 1121.262,A -85,B 0,C 180,E1 16866.048,E2 16866.048} C_VEL
LIN {X 0,Y 411.577,Z 1138.623,A -85,B 0,C 180,E1 16863.467,E2 16863.467} C_VEL
LIN {X 0,Y 407.383,Z 1152.771,A -85,B 0,C 180,E1 16861.025,E2 16861.025} C_VEL
LIN {X 0,Y 402.949,Z 1168.024,A -85,B 0,C 180,E1 16857.946,E2 16857.946} C_VEL
LIN {X 0,Y 399.594,Z 1180.395,A -85,B 0,C 180,E1 16855.016,E2 16855.016} C_VEL
LIN {X 0,Y 396.695,Z 1191.993,A -85,B 0,C 180,E1 16851.747,E2 16851.747} C_VEL
LIN {X 0,Y 394.683,Z 1201.367,A -85,B 0,C 180,E1 16848.614,E2 16848.614} C_VEL
LIN {X 0,Y 393.215,Z 1209.693,A -85,B 0,C 180,E1 16845.183,E2 16845.183} C_VEL
LIN {X 0,Y 392.464,Z 1215.516,A -85,B 0,C 180,E1 16842.208,E2 16842.208} C_VEL
LIN {X 0,Y 392.06,Z 1220.781,A -85,B 0,C 180,E1 16838.654,E2 16838.654} C_VEL
LIN {X 0,Y 391.944,Z 1223.758,A -85,B 0,C 180,E1 16835.71,E2 16835.71} C_VEL
LIN {X 0,Y 391.932,Z 1225.56,A -85,B 0,C 180,E1 16832.778,E2 16832.778} C_VEL
LIN {X 0,Y 391.943,Z 1226.097,A -85,B 0,C 180,E1 16829.561,E2 16829.561} C_VEL
LIN {X 0,Y 391.94,Z 1225.266,A -85,B 0,C 180,E1 16826.636,E2 16826.636} C_VEL
LIN {X 0,Y 391.964,Z 1223.387,A -85,B 0,C 180,E1 16823.85,E2 16823.85} C_VEL
LIN {X 0,Y 392.117,Z 1219.652,A -85,B 0,C 180,E1 16820.46,E2 16820.46} C_VEL
LIN {X 0,Y 392.566,Z 1214.605,A -85,B 0,C 180,E1 16817.299,E2 16817.299} C_VEL
LIN {X 0,Y 393.481,Z 1208.072,A -85,B 0,C 180,E1 16814.072,E2 16814.072} C_VEL
LIN {X 0,Y 395.021,Z 1199.559,A -85,B 0,C 180,E1 16810.761,E2 16810.761} C_VEL
LIN {X 0,Y 397.15,Z 1190.038,A -85,B 0,C 180,E1 16807.657,E2 16807.657} C_VEL
LIN {X 0,Y 400.16,Z 1178.109,A -85,B 0,C 180,E1 16804.428,E2 16804.428} C_VEL
LIN {X 0,Y 403.752,Z 1165.235,A -85,B 0,C 180,E1 16801.449,E2 16801.449} C_VEL
LIN {X 0,Y 407.831,Z 1151.097,A -85,B 0,C 180,E1 16798.685,E2 16798.685} C_VEL
LIN {X 0,Y 412.374,Z 1135.914,A -85,B 0,C 180,E1 16796.105,E2 16796.105} C_VEL
LIN {X 0,Y 417.429,Z 1118.844,A -85,B 0,C 180,E1 16793.642,E2 16793.642} C_VEL
LIN {X 0,Y 422.569,Z 1101.308,A -85,B 0,C 180,E1 16791.449,E2 16791.449} C_VEL
LIN {X 0,Y 427.847,Z 1082.18,A -85,B 0,C 180,E1 16789.423,E2 16789.423} C_VEL
LIN {X 0,Y 433.086,Z 1062.33,A -85,B 0,C 180,E1 16787.613,E2 16787.613} C_VEL
LIN {X 0,Y 438.166,Z 1040.929,A -85,B 0,C 180,E1 16785.985,E2 16785.985} C_VEL
LIN {X 0,Y 443.017,Z 1018.612,A -85,B 0,C 180,E1 16784.561,E2 16784.561} C_VEL
LIN {X 0,Y 446.944,Z 997.493,A -85,B 0,C 180,E1 16783.453,E2 16783.453} C_VEL
LIN {X 0,Y 450.761,Z 973.698,A -85,B 0,C 180,E1 16782.437,E2 16782.437} C_VEL
LIN {X 0,Y 453.666,Z 950.992,A -85,B 0,C 180,E1 16781.693,E2 16781.693} C_VEL
LIN {X 0,Y 456.129,Z 925.18,A -85,B 0,C 180,E1 16781.07,E2 16781.07} C_VEL
LIN {X 0,Y 467.982,Z 707.032,A -85,B 0,C 180,E1 16777.365,E2 16777.365} C_VEL
LIN {X 0,Y 471.529,Z 640.142,A -85,B 0,C 180,E1 16776.235,E2 16776.235} C_VEL
LIN {X 0,Y 459.925,Z 621.598,A -85,B 0,C 180,E1 16773.968,E2 16773.968} C_VEL
LIN {X 0,Y 448.421,Z 604.857,A -85,B 0,C 180,E1 16771.526,E2 16771.526} C_VEL
LIN {X 0,Y 437.516,Z 590.255,A -85,B 0,C 180,E1 16768.98,E2 16768.98} C_VEL
LIN {X 0,Y 428.052,Z 578.601,A -85,B 0,C 180,E1 16766.535,E2 16766.535} C_VEL
LIN {X 0,Y 419.993,Z 568.932,A -85,B 0,C 180,E1 16764.173,E2 16764.173} C_VEL
LIN {X 0,Y 417.872,Z 564.829,A -85,B 0,C 180,E1 16762.659,E2 16762.659} C_VEL
LIN {X 0,Y 415.599,Z 560.431,A -85,B 0,C 180,E1 16760.859,E2 16760.859} C_VEL
LIN {X 0,Y 413.369,Z 556.102,A -85,B 0,C 180,E1 16758.913,E2 16758.913} C_VEL
LIN {X 0,Y 411.18,Z 552.019,A -85,B 0,C 180,E1 16756.821,E2 16756.821} C_VEL
LIN {X 0,Y 408.203,Z 546.585,A -85,B 0,C 180,E1 16753.489,E2 16753.489} C_VEL
LIN {X 0,Y 404.884,Z 540.893,A -85,B 0,C 180,E1 16748.521,E2 16748.521} C_VEL
LIN {X 0,Y 402.583,Z 537.903,A -85,B 0,C 180,E1 16742.705,E2 16742.705} C_VEL
LIN {X 0,Y 402.397,Z 537.403,A -85,B 0,C 180,E1 16739.003,E2 16739.003} C_VEL
LIN {X 0,Y 403.028,Z 538.74,A -85,B 0,C 180,E1 16734.733,E2 16734.733} C_VEL
LIN {X 0,Y 405.112,Z 541.289,A -85,B 0,C 180,E1 16730.481,E2 16730.481} C_VEL
LIN {X 0,Y 407.775,Z 546.037,A -85,B 0,C 180,E1 16726.385,E2 16726.385} C_VEL
LIN {X 0,Y 410.559,Z 551.074,A -85,B 0,C 180,E1 16723.153,E2 16723.153} C_VEL
LIN {X 0,Y 413.727,Z 557.051,A -85,B 0,C 180,E1 16720.068,E2 16720.068} C_VEL
LIN {X 0,Y 416.335,Z 562.065,A -85,B 0,C 180,E1 16717.848,E2 16717.848} C_VEL
LIN {X 0,Y 418.987,Z 567.389,A -85,B 0,C 180,E1 16715.766,E2 16715.766} C_VEL
LIN {X 0,Y 422.58,Z 574.313,A -85,B 0,C 180,E1 16713.284,E2 16713.284} C_VEL
LIN {X 0,Y 428.323,Z 586.637,A -85,B 0,C 180,E1 16709.564,E2 16709.564} C_VEL
LIN {X 0,Y 433.853,Z 599.515,A -85,B 0,C 180,E1 16706.26,E2 16706.26} C_VEL
LIN {X 0,Y 439.247,Z 613.056,A -85,B 0,C 180,E1 16703.224,E2 16703.224} C_VEL
LIN {X 0,Y 440.776,Z 616.36,A -85,B 0,C 180,E1 16702.64,E2 16702.64} C_VEL
LIN {X 0,Y 450.097,Z 631.78,A -85,B 0,C 180,E1 16700.513,E2 16700.513} C_VEL
LIN {X 0,Y 456.816,Z 643.809,A -85,B 0,C 180,E1 16699.075,E2 16699.075} C_VEL
LIN {X 0,Y 463.008,Z 693.712,A -85,B 0,C 180,E1 16696.943,E2 16696.943} C_VEL
LIN {X 0,Y 465.349,Z 715.145,A -85,B 0,C 180,E1 16696.124,E2 16696.124} C_VEL
LIN {X 0,Y 455.229,Z 949.003,A -85,B 0,C 180,E1 16692.561,E2 16692.561} C_VEL
LIN {X 0,Y 453.057,Z 971.671,A -85,B 0,C 180,E1 16692.051,E2 16692.051} C_VEL
LIN {X 0,Y 450.211,Z 992.885,A -85,B 0,C 180,E1 16691.396,E2 16691.396} C_VEL
LIN {X 0,Y 446.721,Z 1013.18,A -85,B 0,C 180,E1 16690.557,E2 16690.557} C_VEL
LIN {X 0,Y 442.335,Z 1034.723,A -85,B 0,C 180,E1 16689.433,E2 16689.433} C_VEL
LIN {X 0,Y 437.912,Z 1053.471,A -85,B 0,C 180,E1 16688.225,E2 16688.225} C_VEL
LIN {X 0,Y 432.861,Z 1072.408,A -85,B 0,C 180,E1 16686.745,E2 16686.745} C_VEL
LIN {X 0,Y 427.558,Z 1090.705,A -85,B 0,C 180,E1 16685.037,E2 16685.037} C_VEL
LIN {X 0,Y 422.273,Z 1107.369,A -85,B 0,C 180,E1 16683.159,E2 16683.159} C_VEL
LIN {X 0,Y 416.644,Z 1124.245,A -85,B 0,C 180,E1 16680.901,E2 16680.901} C_VEL
LIN {X 0,Y 411.645,Z 1138.773,A -85,B 0,C 180,E1 16678.587,E2 16678.587} C_VEL
LIN {X 0,Y 407.02,Z 1151.885,A -85,B 0,C 180,E1 16676.086,E2 16676.086} C_VEL
LIN {X 0,Y 402.908,Z 1163.835,A -85,B 0,C 180,E1 16673.394,E2 16673.394} C_VEL
LIN {X 0,Y 399.38,Z 1174.367,A -85,B 0,C 180,E1 16670.517,E2 16670.517} C_VEL
LIN {X 0,Y 396.423,Z 1183.955,A -85,B 0,C 180,E1 16667.315,E2 16667.315} C_VEL
LIN {X 0,Y 394.44,Z 1191.409,A -85,B 0,C 180,E1 16664.234,E2 16664.234} C_VEL
LIN {X 0,Y 393.083,Z 1197.48,A -85,B 0,C 180,E1 16660.925,E2 16660.925} C_VEL
LIN {X 0,Y 392.332,Z 1202.07,A -85,B 0,C 180,E1 16657.468,E2 16657.468} C_VEL
LIN {X 0,Y 392.065,Z 1204.772,A -85,B 0,C 180,E1 16654.303,E2 16654.303} C_VEL
LIN {X 0,Y 391.983,Z 1205.957,A -85,B 0,C 180,E1 16651.169,E2 16651.169} C_VEL
LIN {X 0,Y 391.992,Z 1205.868,A -85,B 0,C 180,E1 16648.1,E2 16648.1} C_VEL
LIN {X 0,Y 392.096,Z 1204.253,A -85,B 0,C 180,E1 16644.879,E2 16644.879} C_VEL
LIN {X 0,Y 392.457,Z 1201.258,A -85,B 0,C 180,E1 16641.65,E2 16641.65} C_VEL
LIN {X 0,Y 393.268,Z 1196.568,A -85,B 0,C 180,E1 16638.413,E2 16638.413} C_VEL
LIN {X 0,Y 394.793,Z 1189.973,A -85,B 0,C 180,E1 16635.029,E2 16635.029} C_VEL
LIN {X 0,Y 396.495,Z 1183.78,A -85,B 0,C 180,E1 16632.513,E2 16632.513} C_VEL
LIN {X 0,Y 396.382,Z 1181.053,A -85,B 0,C 180,E1 16631.464,E2 16631.464} C_VEL
LIN {X 0,Y 392.961,Z 1173.349,A -85,B 0,C 180,E1 16628.631,E2 16628.631} C_VEL
LIN {X 0,Y 393.232,Z 1170.533,A -85,B 0,C 180,E1 16627.75,E2 16627.75} C_VEL
LIN {X 0,Y 397.284,Z 1159.073,A -85,B 0,C 180,E1 16624.829,E2 16624.829} C_VEL
LIN {X 0,Y 402.196,Z 1145.619,A -85,B 0,C 180,E1 16621.975,E2 16621.975} C_VEL
LIN {X 0,Y 407.272,Z 1131.704,A -85,B 0,C 180,E1 16619.513,E2 16619.513} C_VEL
LIN {X 0,Y 412.56,Z 1116.654,A -85,B 0,C 180,E1 16617.286,E2 16617.286} C_VEL
LIN {X 0,Y 418.14,Z 1100.259,A -85,B 0,C 180,E1 16615.229,E2 16615.229} C_VEL
LIN {X 0,Y 423.596,Z 1082.894,A -85,B 0,C 180,E1 16613.416,E2 16613.416} C_VEL
LIN {X 0,Y 429.258,Z 1063.332,A -85,B 0,C 180,E1 16611.714,E2 16611.714} C_VEL
LIN {X 0,Y 434.377,Z 1043.696,A -85,B 0,C 180,E1 16610.301,E2 16610.301} C_VEL
LIN {X 0,Y 438.799,Z 1023.989,A -85,B 0,C 180,E1 16609.159,E2 16609.159} C_VEL
LIN {X 0,Y 442.976,Z 1002.377,A -85,B 0,C 180,E1 16608.149,E2 16608.149} C_VEL
LIN {X 0,Y 446.241,Z 981.516,A -85,B 0,C 180,E1 16607.401,E2 16607.401} C_VEL
LIN {X 0,Y 448.925,Z 958.74,A -85,B 0,C 180,E1 16606.807,E2 16606.807} C_VEL
LIN {X 0,Y 450.526,Z 935.718,A -85,B 0,C 180,E1 16606.378,E2 16606.378} C_VEL
LIN {X 0,Y 460.201,Z 714.808,A -85,B 0,C 180,E1 16602.99,E2 16602.99} C_VEL
LIN {X 0,Y 453.907,Z 660.685,A -85,B 0,C 180,E1 16600.726,E2 16600.726} C_VEL
LIN {X 0,Y 452.159,Z 647.795,A -85,B 0,C 180,E1 16600.116,E2 16600.116} C_VEL
LIN {X 0,Y 442.848,Z 631.483,A -85,B 0,C 180,E1 16598.031,E2 16598.031} C_VEL
LIN {X 0,Y 433.27,Z 615.901,A -85,B 0,C 180,E1 16595.695,E2 16595.695} C_VEL
LIN {X 0,Y 431.341,Z 612.376,A -85,B 0,C 180,E1 16595.089,E2 16595.089} C_VEL
LIN {X 0,Y 426.172,Z 599.667,A -85,B 0,C 180,E1 16592.022,E2 16592.022} C_VEL
LIN {X 0,Y 421.089,Z 588.131,A -85,B 0,C 180,E1 16588.816,E2 16588.816} C_VEL
LIN {X 0,Y 416.579,Z 578.661,A -85,B 0,C 180,E1 16585.75,E2 16585.75} C_VEL
LIN {X 0,Y 413.092,Z 571.419,A -85,B 0,C 180,E1 16583.087,E2 16583.087} C_VEL
LIN {X 0,Y 410.505,Z 566.475,A -85,B 0,C 180,E1 16580.981,E2 16580.981} C_VEL
LIN {X 0,Y 408.196,Z 561.987,A -85,B 0,C 180,E1 16578.865,E2 16578.865} C_VEL
LIN {X 0,Y 405.878,Z 557.509,A -85,B 0,C 180,E1 16576.458,E2 16576.458} C_VEL
LIN {X 0,Y 403.071,Z 552.403,A -85,B 0,C 180,E1 16573.047,E2 16573.047} C_VEL
LIN {X 0,Y 400.364,Z 547.469,A -85,B 0,C 180,E1 16568.473,E2 16568.473} C_VEL
LIN {X 0,Y 398.349,Z 544.851,A -85,B 0,C 180,E1 16562.878,E2 16562.878} C_VEL
LIN {X 0,Y 398.199,Z 544.521,A -85,B 0,C 180,E1 16559.281,E2 16559.281} C_VEL
LIN {X 0,Y 398.964,Z 545.876,A -85,B 0,C 180,E1 16554.968,E2 16554.968} C_VEL
LIN {X 0,Y 400.797,Z 548.068,A -85,B 0,C 180,E1 16551.247,E2 16551.247} C_VEL
LIN {X 0,Y 403.736,Z 553.351,A -85,B 0,C 180,E1 16546.684,E2 16546.684} C_VEL
LIN {X 0,Y 406.007,Z 557.58,A -85,B 0,C 180,E1 16543.989,E2 16543.989} C_VEL
LIN {X 0,Y 407.112,Z 560.046,A -85,B 0,C 180,E1 16542.711,E2 16542.711} C_VEL
LIN {X 0,Y 409.16,Z 563.452,A -85,B 0,C 180,E1 16540.885,E2 16540.885} C_VEL
LIN {X 0,Y 411.735,Z 568.498,A -85,B 0,C 180,E1 16538.637,E2 16538.637} C_VEL
LIN {X 0,Y 413.311,Z 571.271,A -85,B 0,C 180,E1 16537.603,E2 16537.603} C_VEL
LIN {X 0,Y 420.879,Z 580.157,A -85,B 0,C 180,E1 16535.209,E2 16535.209} C_VEL
LIN {X 0,Y 428.86,Z 589.814,A -85,B 0,C 180,E1 16532.958,E2 16532.958} C_VEL
LIN {X 0,Y 438.871,Z 602.683,A -85,B 0,C 180,E1 16530.407,E2 16530.407} C_VEL
LIN {X 0,Y 449.727,Z 618.046,A -85,B 0,C 180,E1 16527.901,E2 16527.901} C_VEL
LIN {X 0,Y 459.667,Z 633.078,A -85,B 0,C 180,E1 16525.804,E2 16525.804} C_VEL
LIN {X 0,Y 466.477,Z 644.285,A -85,B 0,C 180,E1 16524.446,E2 16524.446} C_VEL
LIN {X 0,Y 453.256,Z 880.476,A -85,B 0,C 180,E1 16520.46,E2 16520.46} C_VEL
LIN {X 0,Y 450.337,Z 930.08,A -85,B 0,C 180,E1 16519.58,E2 16519.58} C_VEL
LIN {X 0,Y 447.782,Z 954.208,A -85,B 0,C 180,E1 16518.957,E2 16518.957} C_VEL
LIN {X 0,Y 444.476,Z 978.405,A -85,B 0,C 180,E1 16518.124,E2 16518.124} C_VEL
LIN {X 0,Y 440.801,Z 1000.052,A -85,B 0,C 180,E1 16517.162,E2 16517.162} C_VEL
LIN {X 0,Y 436.087,Z 1023.847,A -85,B 0,C 180,E1 16515.86,E2 16515.86} C_VEL
LIN {X 0,Y 431.447,Z 1044.186,A -85,B 0,C 180,E1 16514.51,E2 16514.51} C_VEL
LIN {X 0,Y 425.826,Z 1066.514,A -85,B 0,C 180,E1 16512.733,E2 16512.733} C_VEL
LIN {X 0,Y 420.928,Z 1084.394,A -85,B 0,C 180,E1 16511.055,E2 16511.055} C_VEL
LIN {X 0,Y 414.946,Z 1104.902,A -85,B 0,C 180,E1 16508.792,E2 16508.792} C_VEL
LIN {X 0,Y 409.826,Z 1121.768,A -85,B 0,C 180,E1 16506.612,E2 16506.612} C_VEL
LIN {X 0,Y 404.391,Z 1139.171,A -85,B 0,C 180,E1 16503.972,E2 16503.972} C_VEL
LIN {X 0,Y 399.806,Z 1154.058,A -85,B 0,C 180,E1 16501.344,E2 16501.344} C_VEL
LIN {X 0,Y 395.432,Z 1168.395,A -85,B 0,C 180,E1 16498.363,E2 16498.363} C_VEL
LIN {X 0,Y 391.934,Z 1180.725,A -85,B 0,C 180,E1 16495.378,E2 16495.378} C_VEL
LIN {X 0,Y 389.022,Z 1191.747,A -85,B 0,C 180,E1 16492.198,E2 16492.198} C_VEL
LIN {X 0,Y 386.969,Z 1200.705,A -85,B 0,C 180,E1 16489.156,E2 16489.156} C_VEL
LIN {X 0,Y 385.377,Z 1209.15,A -85,B 0,C 180,E1 16485.654,E2 16485.654} C_VEL
LIN {X 0,Y 384.545,Z 1215.03,A -85,B 0,C 180,E1 16482.616,E2 16482.616} C_VEL
LIN {X 0,Y 384.081,Z 1220.232,A -85,B 0,C 180,E1 16479.137,E2 16479.137} C_VEL
LIN {X 0,Y 383.957,Z 1223.431,A -85,B 0,C 180,E1 16475.979,E2 16475.979} C_VEL
LIN {X 0,Y 383.937,Z 1225.211,A -85,B 0,C 180,E1 16473.135,E2 16473.135} C_VEL
LIN {X 0,Y 383.956,Z 1225.941,A -85,B 0,C 180,E1 16469.851,E2 16469.851} C_VEL
LIN {X 0,Y 383.94,Z 1225.133,A -85,B 0,C 180,E1 16466.716,E2 16466.716} C_VEL
LIN {X 0,Y 383.963,Z 1223.3,A -85,B 0,C 180,E1 16463.871,E2 16463.871} C_VEL
LIN {X 0,Y 384.105,Z 1219.868,A -85,B 0,C 180,E1 16460.561,E2 16460.561} C_VEL
LIN {X 0,Y 384.597,Z 1214.588,A -85,B 0,C 180,E1 16457.147,E2 16457.147} C_VEL
LIN {X 0,Y 385.545,Z 1208.165,A -85,B 0,C 180,E1 16453.89,E2 16453.89} C_VEL
LIN {X 0,Y 387.161,Z 1199.719,A -85,B 0,C 180,E1 16450.503,E2 16450.503} C_VEL
LIN {X 0,Y 389.256,Z 1190.748,A -85,B 0,C 180,E1 16447.497,E2 16447.497} C_VEL
LIN {X 0,Y 392.4,Z 1178.883,A -85,B 0,C 180,E1 16444.169,E2 16444.169} C_VEL
LIN {X 0,Y 395.85,Z 1166.933,A -85,B 0,C 180,E1 16441.32,E2 16441.32} C_VEL
LIN {X 0,Y 400.505,Z 1151.582,A -85,B 0,C 180,E1 16438.213,E2 16438.213} C_VEL
LIN {X 0,Y 405.218,Z 1136.458,A -85,B 0,C 180,E1 16435.595,E2 16435.595} C_VEL
LIN {X 0,Y 410.457,Z 1119.513,A -85,B 0,C 180,E1 16433.097,E2 16433.097} C_VEL
LIN {X 0,Y 415.629,Z 1102.487,A -85,B 0,C 180,E1 16430.929,E2 16430.929} C_VEL
LIN {X 0,Y 421.319,Z 1082.71,A -85,B 0,C 180,E1 16428.792,E2 16428.792} C_VEL
LIN {X 0,Y 426.656,Z 1063.172,A -85,B 0,C 180,E1 16426.986,E2 16426.986} C_VEL
LIN {X 0,Y 431.853,Z 1042.118,A -85,B 0,C 180,E1 16425.357,E2 16425.357} C_VEL
LIN {X 0,Y 436.78,Z 1020.406,A -85,B 0,C 180,E1 16423.941,E2 16423.941} C_VEL
LIN {X 0,Y 441.114,Z 997.834,A -85,B 0,C 180,E1 16422.744,E2 16422.744} C_VEL
LIN {X 0,Y 445.025,Z 974.202,A -85,B 0,C 180,E1 16421.726,E2 16421.726} C_VEL
LIN {X 0,Y 448.035,Z 951.331,A -85,B 0,C 180,E1 16420.971,E2 16420.971} C_VEL
LIN {X 0,Y 450.556,Z 925.66,A -85,B 0,C 180,E1 16420.347,E2 16420.347} C_VEL
LIN {X 0,Y 462.329,Z 715.351,A -85,B 0,C 180,E1 16416.752,E2 16416.752} C_VEL
LIN {X 0,Y 466.226,Z 643.83,A -85,B 0,C 180,E1 16415.535,E2 16415.535} C_VEL
LIN {X 0,Y 454.945,Z 625.848,A -85,B 0,C 180,E1 16413.255,E2 16413.255} C_VEL
LIN {X 0,Y 444.768,Z 610.908,A -85,B 0,C 180,E1 16411.023,E2 16411.023} C_VEL
LIN {X 0,Y 434.501,Z 596.964,A -85,B 0,C 180,E1 16408.56,E2 16408.56} C_VEL
LIN {X 0,Y 425.501,Z 585.71,A -85,B 0,C 180,E1 16406.18,E2 16406.18} C_VEL
LIN {X 0,Y 417.115,Z 575.706,A -85,B 0,C 180,E1 16403.711,E2 16403.711} C_VEL
LIN {X 0,Y 412.676,Z 570.468,A -85,B 0,C 180,E1 16402.209,E2 16402.209} C_VEL
LIN {X 0,Y 410.763,Z 566.681,A -85,B 0,C 180,E1 16400.669,E2 16400.669} C_VEL
LIN {X 0,Y 408.557,Z 562.397,A -85,B 0,C 180,E1 16398.7,E2 16398.7} C_VEL
LIN {X 0,Y 406.006,Z 557.59,A -85,B 0,C 180,E1 16396.158,E2 16396.158} C_VEL
LIN {X 0,Y 403.7,Z 553.318,A -85,B 0,C 180,E1 16393.463,E2 16393.463} C_VEL
LIN {X 0,Y 400.48,Z 547.565,A -85,B 0,C 180,E1 16388.471,E2 16388.471} C_VEL
LIN {X 0,Y 398.241,Z 544.629,A -85,B 0,C 180,E1 16382.734,E2 16382.734} C_VEL
LIN {X 0,Y 398.05,Z 544.121,A -85,B 0,C 180,E1 16378.992,E2 16378.992} C_VEL
LIN {X 0,Y 398.639,Z 545.407,A -85,B 0,C 180,E1 16374.819,E2 16374.819} C_VEL
LIN {X 0,Y 400.671,Z 547.978,A -85,B 0,C 180,E1 16370.52,E2 16370.52} C_VEL
LIN {X 0,Y 403.634,Z 553.348,A -85,B 0,C 180,E1 16365.95,E2 16365.95} C_VEL
LIN {X 0,Y 405.774,Z 557.397,A -85,B 0,C 180,E1 16363.391,E2 16363.391} C_VEL
LIN {X 0,Y 409.027,Z 563.605,A -85,B 0,C 180,E1 16360.136,E2 16360.136} C_VEL
LIN {X 0,Y 411.466,Z 568.297,A -85,B 0,C 180,E1 16358.023,E2 16358.023} C_VEL
LIN {X 0,Y 414.252,Z 574.003,A -85,B 0,C 180,E1 16355.774,E2 16355.774} C_VEL
LIN {X 0,Y 417.59,Z 580.598,A -85,B 0,C 180,E1 16353.4,E2 16353.4} C_VEL
LIN {X 0,Y 423.047,Z 592.461,A -85,B 0,C 180,E1 16349.772,E2 16349.772} C_VEL
LIN {X 0,Y 428.521,Z 605.425,A -85,B 0,C 180,E1 16346.406,E2 16346.406} C_VEL
LIN {X 0,Y 432.036,Z 613.921,A -85,B 0,C 180,E1 16344.485,E2 16344.485} C_VEL
LIN {X 0,Y 442.505,Z 630.993,A -85,B 0,C 180,E1 16341.912,E2 16341.912} C_VEL
LIN {X 0,Y 452.193,Z 647.978,A -85,B 0,C 180,E1 16339.744,E2 16339.744} C_VEL
LIN {X 0,Y 457.991,Z 696.285,A -85,B 0,C 180,E1 16337.65,E2 16337.65} C_VEL
LIN {X 0,Y 460.118,Z 716.663,A -85,B 0,C 180,E1 16336.861,E2 16336.861} C_VEL
LIN {X 0,Y 449.678,Z 948.69,A -85,B 0,C 180,E1 16333.296,E2 16333.296} C_VEL
LIN {X 0,Y 447.448,Z 971.383,A -85,B 0,C 180,E1 16332.784,E2 16332.784} C_VEL
LIN {X 0,Y 444.544,Z 992.512,A -85,B 0,C 180,E1 16332.13,E2 16332.13} C_VEL
LIN {X 0,Y 440.951,Z 1012.832,A -85,B 0,C 180,E1 16331.288,E2 16331.288} C_VEL
LIN {X 0,Y 436.444,Z 1034.422,A -85,B 0,C 180,E1 16330.158,E2 16330.158} C_VEL
LIN {X 0,Y 431.946,Z 1052.953,A -85,B 0,C 180,E1 16328.96,E2 16328.96} C_VEL
LIN {X 0,Y 426.68,Z 1072.171,A -85,B 0,C 180,E1 16327.452,E2 16327.452} C_VEL
LIN {X 0,Y 421.2,Z 1090.506,A -85,B 0,C 180,E1 16325.73,E2 16325.73} C_VEL
LIN {X 0,Y 415.552,Z 1107.74,A -85,B 0,C 180,E1 16323.766,E2 16323.766} C_VEL
LIN {X 0,Y 409.736,Z 1124.567,A -85,B 0,C 180,E1 16321.481,E2 16321.481} C_VEL
LIN {X 0,Y 404.557,Z 1139.077,A -85,B 0,C 180,E1 16319.136,E2 16319.136} C_VEL
LIN {X 0,Y 399.757,Z 1152.156,A -85,B 0,C 180,E1 16316.597,E2 16316.597} C_VEL
LIN {X 0,Y 395.471,Z 1164.084,A -85,B 0,C 180,E1 16313.861,E2 16313.861} C_VEL
LIN {X 0,Y 391.761,Z 1174.69,A -85,B 0,C 180,E1 16310.909,E2 16310.909} C_VEL
LIN {X 0,Y 388.69,Z 1184.182,A -85,B 0,C 180,E1 16307.67,E2 16307.67} C_VEL
LIN {X 0,Y 386.514,Z 1191.921,A -85,B 0,C 180,E1 16304.379,E2 16304.379} C_VEL
LIN {X 0,Y 385.137,Z 1197.816,A -85,B 0,C 180,E1 16301.076,E2 16301.076} C_VEL
LIN {X 0,Y 384.361,Z 1202.278,A -85,B 0,C 180,E1 16297.624,E2 16297.624} C_VEL
LIN {X 0,Y 384.071,Z 1205.003,A -85,B 0,C 180,E1 16294.359,E2 16294.359} C_VEL
LIN {X 0,Y 383.986,Z 1206.183,A -85,B 0,C 180,E1 16291.044,E2 16291.044} C_VEL
LIN {X 0,Y 384.001,Z 1206.009,A -85,B 0,C 180,E1 16287.762,E2 16287.762} C_VEL
LIN {X 0,Y 384.118,Z 1204.352,A -85,B 0,C 180,E1 16284.623,E2 16284.623} C_VEL
LIN {X 0,Y 384.518,Z 1201.273,A -85,B 0,C 180,E1 16281.326,E2 16281.326} C_VEL
LIN {X 0,Y 385.411,Z 1196.539,A -85,B 0,C 180,E1 16278.022,E2 16278.022} C_VEL
LIN {X 0,Y 387.065,Z 1189.855,A -85,B 0,C 180,E1 16274.57,E2 16274.57} C_VEL
LIN {X 0,Y 389.507,Z 1181.705,A -85,B 0,C 180,E1 16271.284,E2 16271.284} C_VEL
LIN {X 0,Y 392.71,Z 1171.979,A -85,B 0,C 180,E1 16268.178,E2 16268.178} C_VEL
LIN {X 0,Y 393.232,Z 1170.533,A -85,B 0,C 180,E1 16267.75,E2 16267.75} C_VEL
LIN {X 0,Y 393.522,Z 1167.181,A -85,B 0,C 180,E1 16266.729,E2 16266.729} C_VEL
LIN {X 0,Y 391.306,Z 1158.275,A -85,B 0,C 180,E1 16264.112,E2 16264.112} C_VEL
LIN {X 0,Y 391.904,Z 1154.215,A -85,B 0,C 180,E1 16263.148,E2 16263.148} C_VEL
LIN {X 0,Y 396.771,Z 1141.411,A -85,B 0,C 180,E1 16260.568,E2 16260.568} C_VEL
LIN {X 0,Y 402.373,Z 1126.396,A -85,B 0,C 180,E1 16258.043,E2 16258.043} C_VEL
LIN {X 0,Y 408.159,Z 1110.467,A -85,B 0,C 180,E1 16255.792,E2 16255.792} C_VEL
LIN {X 0,Y 413.705,Z 1094.097,A -85,B 0,C 180,E1 16253.864,E2 16253.864} C_VEL
LIN {X 0,Y 419.713,Z 1075.075,A -85,B 0,C 180,E1 16251.989,E2 16251.989} C_VEL
LIN {X 0,Y 425.269,Z 1055.852,A -85,B 0,C 180,E1 16250.42,E2 16250.42} C_VEL
LIN {X 0,Y 430.165,Z 1036.43,A -85,B 0,C 180,E1 16249.133,E2 16249.133} C_VEL
LIN {X 0,Y 434.794,Z 1015.455,A -85,B 0,C 180,E1 16247.996,E2 16247.996} C_VEL
LIN {X 0,Y 438.451,Z 995.573,A -85,B 0,C 180,E1 16247.146,E2 16247.146} C_VEL
LIN {X 0,Y 441.823,Z 972.717,A -85,B 0,C 180,E1 16246.406,E2 16246.406} C_VEL
LIN {X 0,Y 444.2,Z 950.26,A -85,B 0,C 180,E1 16245.88,E2 16245.88} C_VEL
LIN {X 0,Y 447.292,Z 885.144,A -85,B 0,C 180,E1 16244.85,E2 16244.85} C_VEL
LIN {X 0,Y 455.045,Z 716.103,A -85,B 0,C 180,E1 16242.228,E2 16242.228} C_VEL
LIN {X 0,Y 448.997,Z 662.206,A -85,B 0,C 180,E1 16239.935,E2 16239.935} C_VEL
LIN {X 0,Y 447.664,Z 652.333,A -85,B 0,C 180,E1 16239.454,E2 16239.454} C_VEL
LIN {X 0,Y 438.429,Z 635.928,A -85,B 0,C 180,E1 16237.306,E2 16237.306} C_VEL
LIN {X 0,Y 428.292,Z 619.279,A -85,B 0,C 180,E1 16234.726,E2 16234.726} C_VEL
LIN {X 0,Y 423.108,Z 611.011,A -85,B 0,C 180,E1 16233.223,E2 16233.223} C_VEL
LIN {X 0,Y 417.79,Z 598.234,A -85,B 0,C 180,E1 16229.855,E2 16229.855} C_VEL
LIN {X 0,Y 412.47,Z 586.423,A -85,B 0,C 180,E1 16226.18,E2 16226.18} C_VEL
LIN {X 0,Y 408.204,Z 577.646,A -85,B 0,C 180,E1 16222.922,E2 16222.922} C_VEL
LIN {X 0,Y 405.659,Z 572.711,A -85,B 0,C 180,E1 16220.79,E2 16220.79} C_VEL
LIN {X 0,Y 403.56,Z 568.487,A -85,B 0,C 180,E1 16218.79,E2 16218.79} C_VEL
LIN {X 0,Y 401.104,Z 563.835,A -85,B 0,C 180,E1 16216.213,E2 16216.213} C_VEL
LIN {X 0,Y 398.5,Z 558.93,A -85,B 0,C 180,E1 16212.904,E2 16212.904} C_VEL
LIN {X 0,Y 395.948,Z 554.134,A -85,B 0,C 180,E1 16208.422,E2 16208.422} C_VEL
LIN {X 0,Y 394.001,Z 551.579,A -85,B 0,C 180,E1 16202.909,E2 16202.909} C_VEL
LIN {X 0,Y 393.857,Z 551.241,A -85,B 0,C 180,E1 16199.273,E2 16199.273} C_VEL
LIN {X 0,Y 394.579,Z 552.551,A -85,B 0,C 180,E1 16195.057,E2 16195.057} C_VEL
LIN {X 0,Y 396.379,Z 554.758,A -85,B 0,C 180,E1 16191.295,E2 16191.295} C_VEL
LIN {X 0,Y 399.185,Z 559.869,A -85,B 0,C 180,E1 16186.824,E2 16186.824} C_VEL
LIN {X 0,Y 401.419,Z 564.094,A -85,B 0,C 180,E1 16184.098,E2 16184.098} C_VEL
LIN {X 0,Y 404.493,Z 570.039,A -85,B 0,C 180,E1 16180.956,E2 16180.956} C_VEL
LIN {X 0,Y 406.01,Z 572.846,A -85,B 0,C 180,E1 16179.756,E2 16179.756} C_VEL
LIN {X 0,Y 413.217,Z 581.083,A -85,B 0,C 180,E1 16177.222,E2 16177.222} C_VEL
LIN {X 0,Y 421.338,Z 590.7,A -85,B 0,C 180,E1 16174.712,E2 16174.712} C_VEL
LIN {X 0,Y 430.069,Z 601.849,A -85,B 0,C 180,E1 16172.29,E2 16172.29} C_VEL
LIN {X 0,Y 439.007,Z 613.856,A -85,B 0,C 180,E1 16170.042,E2 16170.042} C_VEL
LIN {X 0,Y 450.049,Z 629.926,A -85,B 0,C 180,E1 16167.513,E2 16167.513} C_VEL
LIN {X 0,Y 461.063,Z 647.55,A -85,B 0,C 180,E1 16165.204,E2 16165.204} C_VEL
LIN {X 0,Y 461.215,Z 648.845,A -85,B 0,C 180,E1 16165.146,E2 16165.146} C_VEL
LIN {X 0,Y 447.644,Z 884.59,A -85,B 0,C 180,E1 16161.145,E2 16161.145} C_VEL
LIN {X 0,Y 444.826,Z 930.607,A -85,B 0,C 180,E1 16160.32,E2 16160.32} C_VEL
LIN {X 0,Y 442.221,Z 954.552,A -85,B 0,C 180,E1 16159.697,E2 16159.697} C_VEL
LIN {X 0,Y 438.914,Z 978.178,A -85,B 0,C 180,E1 16158.882,E2 16158.882} C_VEL
LIN {X 0,Y 435.138,Z 999.843,A -85,B 0,C 180,E1 16157.918,E2 16157.918} C_VEL
LIN {X 0,Y 430.653,Z 1022.121,A -85,B 0,C 180,E1 16156.707,E2 16156.707} C_VEL
LIN {X 0,Y 425.841,Z 1042.641,A -85,B 0,C 180,E1 16155.351,E2 16155.351} C_VEL
LIN {X 0,Y 420.433,Z 1063.752,A -85,B 0,C 180,E1 16153.698,E2 16153.698} C_VEL
LIN {X 0,Y 414.897,Z 1083.315,A -85,B 0,C 180,E1 16151.868,E2 16151.868} C_VEL
LIN {X 0,Y 408.886,Z 1103.373,A -85,B 0,C 180,E1 16149.66,E2 16149.66} C_VEL
LIN {X 0,Y 403.703,Z 1119.788,A -85,B 0,C 180,E1 16147.537,E2 16147.537} C_VEL
LIN {X 0,Y 397.813,Z 1137.98,A -85,B 0,C 180,E1 16144.788,E2 16144.788} C_VEL
LIN {X 0,Y 392.97,Z 1152.956,A -85,B 0,C 180,E1 16142.125,E2 16142.125} C_VEL
LIN {X 0,Y 388.377,Z 1167.382,A -85,B 0,C 180,E1 16139.115,E2 16139.115} C_VEL
LIN {X 0,Y 384.779,Z 1179.268,A -85,B 0,C 180,E1 16136.215,E2 16136.215} C_VEL
LIN {X 0,Y 381.495,Z 1191.023,A -85,B 0,C 180,E1 16132.823,E2 16132.823} C_VEL
LIN {X 0,Y 379.285,Z 1200.044,A -85,B 0,C 180,E1 16129.72,E2 16129.72} C_VEL
LIN {X 0,Y 377.475,Z 1209.029,A -85,B 0,C 180,E1 16125.94,E2 16125.94} C_VEL
LIN {X 0,Y 376.602,Z 1214.811,A -85,B 0,C 180,E1 16122.886,E2 16122.886} C_VEL
LIN {X 0,Y 376.095,Z 1220.021,A -85,B 0,C 180,E1 16119.333,E2 16119.333} C_VEL
LIN {X 0,Y 375.963,Z 1223.224,A -85,B 0,C 180,E1 16116.107,E2 16116.107} C_VEL
LIN {X 0,Y 375.94,Z 1225.006,A -85,B 0,C 180,E1 16113.202,E2 16113.202} C_VEL
LIN {X 0,Y 375.959,Z 1225.736,A -85,B 0,C 180,E1 16109.848,E2 16109.848} C_VEL
LIN {X 0,Y 375.943,Z 1224.927,A -85,B 0,C 180,E1 16106.646,E2 16106.646} C_VEL
LIN {X 0,Y 375.969,Z 1223.092,A -85,B 0,C 180,E1 16103.74,E2 16103.74} C_VEL
LIN {X 0,Y 376.14,Z 1219.439,A -85,B 0,C 180,E1 16100.205,E2 16100.205} C_VEL
LIN {X 0,Y 376.635,Z 1214.52,A -85,B 0,C 180,E1 16096.959,E2 16096.959} C_VEL
LIN {X 0,Y 377.611,Z 1208.259,A -85,B 0,C 180,E1 16093.7,E2 16093.7} C_VEL
LIN {X 0,Y 379.377,Z 1199.579,A -85,B 0,C 180,E1 16090.124,E2 16090.124} C_VEL
LIN {X 0,Y 381.62,Z 1190.501,A -85,B 0,C 180,E1 16087.022,E2 16087.022} C_VEL
LIN {X 0,Y 384.941,Z 1178.615,A -85,B 0,C 180,E1 16083.63,E2 16083.63} C_VEL
LIN {X 0,Y 388.593,Z 1166.624,A -85,B 0,C 180,E1 16080.725,E2 16080.725} C_VEL
LIN {X 0,Y 393.206,Z 1152.07,A -85,B 0,C 180,E1 16077.724,E2 16077.724} C_VEL
LIN {X 0,Y 398.096,Z 1137.006,A -85,B 0,C 180,E1 16075.065,E2 16075.065} C_VEL
LIN {X 0,Y 403.687,Z 1119.663,A -85,B 0,C 180,E1 16072.461,E2 16072.461} C_VEL
LIN {X 0,Y 409.049,Z 1102.659,A -85,B 0,C 180,E1 16070.268,E2 16070.268} C_VEL
LIN {X 0,Y 414.895,Z 1083.063,A -85,B 0,C 180,E1 16068.122,E2 16068.122} C_VEL
LIN {X 0,Y 420.378,Z 1063.667,A -85,B 0,C 180,E1 16066.31,E2 16066.31} C_VEL
LIN {X 0,Y 425.817,Z 1042.394,A -85,B 0,C 180,E1 16064.645,E2 16064.645} C_VEL
LIN {X 0,Y 430.868,Z 1020.821,A -85,B 0,C 180,E1 16063.226,E2 16063.226} C_VEL
LIN {X 0,Y 435.354,Z 998.186,A -85,B 0,C 180,E1 16062.015,E2 16062.015} C_VEL
LIN {X 0,Y 439.361,Z 974.719,A -85,B 0,C 180,E1 16060.996,E2 16060.996} C_VEL
LIN {X 0,Y 442.47,Z 951.737,A -85,B 0,C 180,E1 16060.233,E2 16060.233} C_VEL
LIN {X 0,Y 445.05,Z 926.273,A -85,B 0,C 180,E1 16059.608,E2 16059.608} C_VEL
LIN {X 0,Y 456.913,Z 720.493,A -85,B 0,C 180,E1 16056.071,E2 16056.071} C_VEL
LIN {X 0,Y 461.009,Z 647.583,A -85,B 0,C 180,E1 16054.822,E2 16054.822} C_VEL
LIN {X 0,Y 449.801,Z 629.594,A -85,B 0,C 180,E1 16052.469,E2 16052.469} C_VEL
LIN {X 0,Y 438.161,Z 612.661,A -85,B 0,C 180,E1 16049.796,E2 16049.796} C_VEL
LIN {X 0,Y 427.792,Z 598.809,A -85,B 0,C 180,E1 16047.153,E2 16047.153} C_VEL
LIN {X 0,Y 418.547,Z 587.43,A -85,B 0,C 180,E1 16044.525,E2 16044.525} C_VEL
LIN {X 0,Y 410.718,Z 578.156,A -85,B 0,C 180,E1 16042.019,E2 16042.019} C_VEL
LIN {X 0,Y 405.648,Z 572.418,A -85,B 0,C 180,E1 16040.187,E2 16040.187} C_VEL
LIN {X 0,Y 403.735,Z 568.657,A -85,B 0,C 180,E1 16038.467,E2 16038.467} C_VEL
LIN {X 0,Y 401.416,Z 564.104,A -85,B 0,C 180,E1 16036.051,E2 16036.051} C_VEL
LIN {X 0,Y 399.077,Z 559.564,A -85,B 0,C 180,E1 16033.179,E2 16033.179} C_VEL
LIN {X 0,Y 395.982,Z 554.148,A -85,B 0,C 180,E1 16028.275,E2 16028.275} C_VEL
LIN {X 0,Y 393.878,Z 551.317,A -85,B 0,C 180,E1 16022.619,E2 16022.619} C_VEL
LIN {X 0,Y 393.702,Z 550.84,A -85,B 0,C 180,E1 16018.981,E2 16018.981} C_VEL
LIN {X 0,Y 394.293,Z 552.151,A -85,B 0,C 180,E1 16014.762,E2 16014.762} C_VEL
LIN {X 0,Y 396.229,Z 554.667,A -85,B 0,C 180,E1 16010.559,E2 16010.559} C_VEL
LIN {X 0,Y 399.063,Z 559.857,A -85,B 0,C 180,E1 16006.082,E2 16006.082} C_VEL
LIN {X 0,Y 401.163,Z 563.901,A -85,B 0,C 180,E1 16003.492,E2 16003.492} C_VEL
LIN {X 0,Y 404.221,Z 569.832,A -85,B 0,C 180,E1 16000.341,E2 16000.341} C_VEL
LIN {X 0,Y 406.743,Z 574.902,A -85,B 0,C 180,E1 15998.058,E2 15998.058} C_VEL
LIN {X 0,Y 410.543,Z 582.355,A -85,B 0,C 180,E1 15995.08,E2 15995.08} C_VEL
LIN {X 0,Y 415.184,Z 592.662,A -85,B 0,C 180,E1 15991.677,E2 15991.677} C_VEL
LIN {X 0,Y 419.552,Z 602.525,A -85,B 0,C 180,E1 15988.821,E2 15988.821} C_VEL
LIN {X 0,Y 423.665,Z 612.137,A -85,B 0,C 180,E1 15986.404,E2 15986.404} C_VEL
LIN {X 0,Y 433.562,Z 627.905,A -85,B 0,C 180,E1 15983.753,E2 15983.753} C_VEL
LIN {X 0,Y 442.885,Z 643.838,A -85,B 0,C 180,E1 15981.497,E2 15981.497} C_VEL
LIN {X 0,Y 447.743,Z 652.823,A -85,B 0,C 180,E1 15980.389,E2 15980.389} C_VEL
LIN {X 0,Y 453.483,Z 702.8,A -85,B 0,C 180,E1 15978.206,E2 15978.206} C_VEL
LIN {X 0,Y 454.969,Z 718.059,A -85,B 0,C 180,E1 15977.615,E2 15977.615} C_VEL
LIN {X 0,Y 444.201,Z 948.369,A -85,B 0,C 180,E1 15974.05,E2 15974.05} C_VEL
LIN {X 0,Y 441.917,Z 971.054,A -85,B 0,C 180,E1 15973.535,E2 15973.535} C_VEL
LIN {X 0,Y 438.819,Z 992.878,A -85,B 0,C 180,E1 15972.854,E2 15972.854} C_VEL
LIN {X 0,Y 435.257,Z 1012.483,A -85,B 0,C 180,E1 15972.038,E2 15972.038} C_VEL
LIN {X 0,Y 430.624,Z 1034.12,A -85,B 0,C 180,E1 15970.902,E2 15970.902} C_VEL
LIN {X 0,Y 426.159,Z 1052.025,A -85,B 0,C 180,E1 15969.743,E2 15969.743} C_VEL
LIN {X 0,Y 420.567,Z 1071.934,A -85,B 0,C 180,E1 15968.179,E2 15968.179} C_VEL
LIN {X 0,Y 414.908,Z 1090.302,A -85,B 0,C 180,E1 15966.443,E2 15966.443} C_VEL
LIN {X 0,Y 409.064,Z 1107.566,A -85,B 0,C 180,E1 15964.461,E2 15964.461} C_VEL
LIN {X 0,Y 402.872,Z 1124.883,A -85,B 0,C 180,E1 15962.08,E2 15962.08} C_VEL
LIN {X 0,Y 397.508,Z 1139.378,A -85,B 0,C 180,E1 15959.704,E2 15959.704} C_VEL
LIN {X 0,Y 392.525,Z 1152.428,A -85,B 0,C 180,E1 15957.126,E2 15957.126} C_VEL
LIN {X 0,Y 387.848,Z 1164.883,A -85,B 0,C 180,E1 15954.198,E2 15954.198} C_VEL
LIN {X 0,Y 384.049,Z 1175.344,A -85,B 0,C 180,E1 15951.216,E2 15951.216} C_VEL
LIN {X 0,Y 380.971,Z 1184.409,A -85,B 0,C 180,E1 15948.041,E2 15948.041} C_VEL
LIN {X 0,Y 378.675,Z 1192.137,A -85,B 0,C 180,E1 15944.683,E2 15944.683} C_VEL
LIN {X 0,Y 377.216,Z 1198.03,A -85,B 0,C 180,E1 15941.312,E2 15941.312} C_VEL
LIN {X 0,Y 376.382,Z 1202.54,A -85,B 0,C 180,E1 15937.731,E2 15937.731} C_VEL
LIN {X 0,Y 376.077,Z 1205.235,A -85,B 0,C 180,E1 15934.416,E2 15934.416} C_VEL
LIN {X 0,Y 375.989,Z 1206.387,A -85,B 0,C 180,E1 15931.067,E2 15931.067} C_VEL
LIN {X 0,Y 376.001,Z 1206.255,A -85,B 0,C 180,E1 15927.866,E2 15927.866} C_VEL
LIN {X 0,Y 376.131,Z 1204.557,A -85,B 0,C 180,E1 15924.509,E2 15924.509} C_VEL
LIN {X 0,Y 376.56,Z 1201.483,A -85,B 0,C 180,E1 15921.141,E2 15921.141} C_VEL
LIN {X 0,Y 377.511,Z 1196.751,A -85,B 0,C 180,E1 15917.767,E2 15917.767} C_VEL
LIN {X 0,Y 379.285,Z 1189.987,A -85,B 0,C 180,E1 15914.204,E2 15914.204} C_VEL
LIN {X 0,Y 381.828,Z 1181.936,A -85,B 0,C 180,E1 15910.894,E2 15910.894} C_VEL
LIN {X 0,Y 385.184,Z 1172.215,A -85,B 0,C 180,E1 15907.729,E2 15907.729} C_VEL
LIN {X 0,Y 389.496,Z 1160.554,A -85,B 0,C 180,E1 15904.615,E2 15904.615} C_VEL
LIN {X 0,Y 391.904,Z 1154.215,A -85,B 0,C 180,E1 15903.148,E2 15903.148} C_VEL
LIN {X 0,Y 392.584,Z 1150.116,A -85,B 0,C 180,E1 15902.195,E2 15902.195} C_VEL
LIN {X 0,Y 391.434,Z 1139.055,A -85,B 0,C 180,E1 15899.551,E2 15899.551} C_VEL
LIN {X 0,Y 392.347,Z 1134.996,A -85,B 0,C 180,E1 15898.784,E2 15898.784} C_VEL
LIN {X 0,Y 398.178,Z 1119.797,A -85,B 0,C 180,E1 15896.379,E2 15896.379} C_VEL
LIN {X 0,Y 404.023,Z 1103.77,A -85,B 0,C 180,E1 15894.265,E2 15894.265} C_VEL
LIN {X 0,Y 410.174,Z 1085.722,A -85,B 0,C 180,E1 15892.277,E2 15892.277} C_VEL
LIN {X 0,Y 415.915,Z 1067.58,A -85,B 0,C 180,E1 15890.606,E2 15890.606} C_VEL
LIN {X 0,Y 421.248,Z 1048.456,A -85,B 0,C 180,E1 15889.163,E2 15889.163} C_VEL
LIN {X 0,Y 426.383,Z 1027.796,A -85,B 0,C 180,E1 15887.882,E2 15887.882} C_VEL
LIN {X 0,Y 430.7,Z 1007.38,A -85,B 0,C 180,E1 15886.869,E2 15886.869} C_VEL
LIN {X 0,Y 434.51,Z 985.32,A -85,B 0,C 180,E1 15886.024,E2 15886.024} C_VEL
LIN {X 0,Y 437.521,Z 963.187,A -85,B 0,C 180,E1 15885.394,E2 15885.394} C_VEL
LIN {X 0,Y 439.376,Z 940.833,A -85,B 0,C 180,E1 15884.948,E2 15884.948} C_VEL
LIN {X 0,Y 449.999,Z 717.658,A -85,B 0,C 180,E1 15881.459,E2 15881.459} C_VEL
LIN {X 0,Y 444.192,Z 663.899,A -85,B 0,C 180,E1 15879.134,E2 15879.134} C_VEL
LIN {X 0,Y 443.239,Z 656.838,A -85,B 0,C 180,E1 15878.777,E2 15878.777} C_VEL
LIN {X 0,Y 434.126,Z 640.5,A -85,B 0,C 180,E1 15876.581,E2 15876.581} C_VEL
LIN {X 0,Y 424.543,Z 624.728,A -85,B 0,C 180,E1 15874.053,E2 15874.053} C_VEL
LIN {X 0,Y 416.445,Z 612.195,A -85,B 0,C 180,E1 15871.683,E2 15871.683} C_VEL
LIN {X 0,Y 414.431,Z 608.691,A -85,B 0,C 180,E1 15870.924,E2 15870.924} C_VEL
LIN {X 0,Y 410.204,Z 598.91,A -85,B 0,C 180,E1 15868.063,E2 15868.063} C_VEL
LIN {X 0,Y 405.643,Z 588.644,A -85,B 0,C 180,E1 15864.619,E2 15864.619} C_VEL
LIN {X 0,Y 401.374,Z 579.766,A -85,B 0,C 180,E1 15861.022,E2 15861.022} C_VEL
LIN {X 0,Y 398.586,Z 574.521,A -85,B 0,C 180,E1 15858.426,E2 15858.426} C_VEL
LIN {X 0,Y 396.491,Z 570.331,A -85,B 0,C 180,E1 15856.098,E2 15856.098} C_VEL
LIN {X 0,Y 394.064,Z 565.596,A -85,B 0,C 180,E1 15852.902,E2 15852.902} C_VEL
LIN {X 0,Y 391.531,Z 560.799,A -85,B 0,C 180,E1 15848.37,E2 15848.37} C_VEL
LIN {X 0,Y 389.641,Z 558.265,A -85,B 0,C 180,E1 15842.795,E2 15842.795} C_VEL
LIN {X 0,Y 389.53,Z 557.973,A -85,B 0,C 180,E1 15839.118,E2 15839.118} C_VEL
LIN {X 0,Y 390.343,Z 559.434,A -85,B 0,C 180,E1 15834.709,E2 15834.709} C_VEL
LIN {X 0,Y 391.961,Z 561.448,A -85,B 0,C 180,E1 15831.344,E2 15831.344} C_VEL
LIN {X 0,Y 394.7,Z 566.649,A -85,B 0,C 180,E1 15826.821,E2 15826.821} C_VEL
LIN {X 0,Y 397.333,Z 571.617,A -85,B 0,C 180,E1 15823.629,E2 15823.629} C_VEL
LIN {X 0,Y 398.895,Z 574.682,A -85,B 0,C 180,E1 15822.117,E2 15822.117} C_VEL
LIN {X 0,Y 405.573,Z 581.986,A -85,B 0,C 180,E1 15819.47,E2 15819.47} C_VEL
LIN {X 0,Y 414.48,Z 592.413,A -85,B 0,C 180,E1 15816.431,E2 15816.431} C_VEL
LIN {X 0,Y 423.943,Z 604.341,A -85,B 0,C 180,E1 15813.603,E2 15813.603} C_VEL
LIN {X 0,Y 433.258,Z 616.757,A -85,B 0,C 180,E1 15811.124,E2 15811.124} C_VEL
LIN {X 0,Y 444.494,Z 633.029,A -85,B 0,C 180,E1 15808.428,E2 15808.428} C_VEL
LIN {X 0,Y 455.453,Z 650.511,A -85,B 0,C 180,E1 15806.032,E2 15806.032} C_VEL
LIN {X 0,Y 456.112,Z 651.943,A -85,B 0,C 180,E1 15805.885,E2 15805.885} C_VEL
LIN {X 0,Y 442.087,Z 888.905,A -85,B 0,C 180,E1 15801.843,E2 15801.843} C_VEL
LIN {X 0,Y 439.38,Z 931.212,A -85,B 0,C 180,E1 15801.075,E2 15801.075} C_VEL
LIN {X 0,Y 436.742,Z 954.848,A -85,B 0,C 180,E1 15800.457,E2 15800.457} C_VEL
LIN {X 0,Y 433.215,Z 979.194,A -85,B 0,C 180,E1 15799.609,E2 15799.609} C_VEL
LIN {X 0,Y 429.342,Z 1000.747,A -85,B 0,C 180,E1 15798.639,E2 15798.639} C_VEL
LIN {X 0,Y 424.341,Z 1024.478,A -85,B 0,C 180,E1 15797.32,E2 15797.32} C_VEL
LIN {X 0,Y 419.48,Z 1044.512,A -85,B 0,C 180,E1 15795.97,E2 15795.97} C_VEL
LIN {X 0,Y 413.425,Z 1067.003,A -85,B 0,C 180,E1 15794.148,E2 15794.148} C_VEL
LIN {X 0,Y 407.801,Z 1086.201,A -85,B 0,C 180,E1 15792.301,E2 15792.301} C_VEL
LIN {X 0,Y 401.795,Z 1105.262,A -85,B 0,C 180,E1 15790.129,E2 15790.129} C_VEL
LIN {X 0,Y 396.311,Z 1122.03,A -85,B 0,C 180,E1 15787.903,E2 15787.903} C_VEL
LIN {X 0,Y 390.417,Z 1139.406,A -85,B 0,C 180,E1 15785.185,E2 15785.185} C_VEL
LIN {X 0,Y 385.188,Z 1155.038,A -85,B 0,C 180,E1 15782.325,E2 15782.325} C_VEL
LIN {X 0,Y 380.468,Z 1169.141,A -85,B 0,C 180,E1 15779.247,E2 15779.247} C_VEL
LIN {X 0,Y 376.489,Z 1181.911,A -85,B 0,C 180,E1 15775.989,E2 15775.989} C_VEL
LIN {X 0,Y 373.356,Z 1192.696,A -85,B 0,C 180,E1 15772.683,E2 15772.683} C_VEL
LIN {X 0,Y 370.971,Z 1202.274,A -85,B 0,C 180,E1 15769.197,E2 15769.197} C_VEL
LIN {X 0,Y 369.441,Z 1209.659,A -85,B 0,C 180,E1 15765.863,E2 15765.863} C_VEL
LIN {X 0,Y 368.487,Z 1215.982,A -85,B 0,C 180,E1 15762.348,E2 15762.348} C_VEL
LIN {X 0,Y 368.07,Z 1220.49,A -85,B 0,C 180,E1 15758.907,E2 15758.907} C_VEL
LIN {X 0,Y 367.956,Z 1223.258,A -85,B 0,C 180,E1 15755.927,E2 15755.927} C_VEL
LIN {X 0,Y 367.943,Z 1225.158,A -85,B 0,C 180,E1 15752.492,E2 15752.492} C_VEL
LIN {X 0,Y 367.952,Z 1225.436,A -85,B 0,C 180,E1 15749.222,E2 15749.222} C_VEL
LIN {X 0,Y 367.95,Z 1224.577,A -85,B 0,C 180,E1 15746.261,E2 15746.261} C_VEL
LIN {X 0,Y 367.986,Z 1222.401,A -85,B 0,C 180,E1 15742.977,E2 15742.977} C_VEL
LIN {X 0,Y 368.219,Z 1218.352,A -85,B 0,C 180,E1 15739.36,E2 15739.36} C_VEL
LIN {X 0,Y 368.814,Z 1213.496,A -85,B 0,C 180,E1 15736.198,E2 15736.198} C_VEL
LIN {X 0,Y 370.156,Z 1205.94,A -85,B 0,C 180,E1 15732.39,E2 15732.39} C_VEL
LIN {X 0,Y 371.945,Z 1198.07,A -85,B 0,C 180,E1 15729.216,E2 15729.216} C_VEL
LIN {X 0,Y 374.742,Z 1187.757,A -85,B 0,C 180,E1 15725.739,E2 15725.739} C_VEL
LIN {X 0,Y 378.075,Z 1176.561,A -85,B 0,C 180,E1 15722.603,E2 15722.603} C_VEL
LIN {X 0,Y 382.485,Z 1162.947,A -85,B 0,C 180,E1 15719.353,E2 15719.353} C_VEL
LIN {X 0,Y 387.138,Z 1148.976,A -85,B 0,C 180,E1 15716.537,E2 15716.537} C_VEL
LIN {X 0,Y 392.863,Z 1132.085,A -85,B 0,C 180,E1 15713.63,E2 15713.63} C_VEL
LIN {X 0,Y 398.17,Z 1116.167,A -85,B 0,C 180,E1 15711.298,E2 15711.298} C_VEL
LIN {X 0,Y 404.414,Z 1096.807,A -85,B 0,C 180,E1 15708.879,E2 15708.879} C_VEL
LIN {X 0,Y 410.017,Z 1078.497,A -85,B 0,C 180,E1 15706.937,E2 15706.937} C_VEL
LIN {X 0,Y 416.035,Z 1057.325,A -85,B 0,C 180,E1 15705.044,E2 15705.044} C_VEL
LIN {X 0,Y 421.025,Z 1038.103,A -85,B 0,C 180,E1 15703.588,E2 15703.588} C_VEL
LIN {X 0,Y 426.249,Z 1015.462,A -85,B 0,C 180,E1 15702.163,E2 15702.163} C_VEL
LIN {X 0,Y 430.403,Z 994.781,A -85,B 0,C 180,E1 15701.086,E2 15701.086} C_VEL
LIN {X 0,Y 434.414,Z 970.93,A -85,B 0,C 180,E1 15700.095,E2 15700.095} C_VEL
LIN {X 0,Y 437.42,Z 948.8,A -85,B 0,C 180,E1 15699.38,E2 15699.38} C_VEL
LIN {X 0,Y 439.83,Z 924.01,A -85,B 0,C 180,E1 15698.796,E2 15698.796} C_VEL
LIN {X 0,Y 453.749,Z 689.019,A -85,B 0,C 180,E1 15694.75,E2 15694.75} C_VEL
LIN {X 0,Y 455.909,Z 651.361,A -85,B 0,C 180,E1 15694.1,E2 15694.1} C_VEL
LIN {X 0,Y 444.975,Z 633.863,A -85,B 0,C 180,E1 15691.723,E2 15691.723} C_VEL
LIN {X 0,Y 434.042,Z 617.923,A -85,B 0,C 180,E1 15689.121,E2 15689.121} C_VEL
LIN {X 0,Y 424.658,Z 605.255,A -85,B 0,C 180,E1 15686.651,E2 15686.651} C_VEL
LIN {X 0,Y 415.892,Z 594.292,A -85,B 0,C 180,E1 15684.087,E2 15684.087} C_VEL
LIN {X 0,Y 408.195,Z 585.105,A -85,B 0,C 180,E1 15681.557,E2 15681.557} C_VEL
LIN {X 0,Y 403.14,Z 579.408,A -85,B 0,C 180,E1 15679.713,E2 15679.713} C_VEL
LIN {X 0,Y 398.564,Z 574.31,A -85,B 0,C 180,E1 15677.841,E2 15677.841} C_VEL
LIN {X 0,Y 396.663,Z 570.425,A -85,B 0,C 180,E1 15675.798,E2 15675.798} C_VEL
LIN {X 0,Y 394.129,Z 565.626,A -85,B 0,C 180,E1 15672.602,E2 15672.602} C_VEL
LIN {X 0,Y 391.576,Z 560.818,A -85,B 0,C 180,E1 15668.221,E2 15668.221} C_VEL
LIN {X 0,Y 389.517,Z 558.006,A -85,B 0,C 180,E1 15662.501,E2 15662.501} C_VEL
LIN {X 0,Y 389.359,Z 557.584,A -85,B 0,C 180,E1 15658.823,E2 15658.823} C_VEL
LIN {X 0,Y 390.029,Z 559.045,A -85,B 0,C 180,E1 15654.409,E2 15654.409} C_VEL
LIN {X 0,Y 391.754,Z 561.177,A -85,B 0,C 180,E1 15650.747,E2 15650.747} C_VEL
LIN {X 0,Y 394.493,Z 566.367,A -85,B 0,C 180,E1 15646.216,E2 15646.216} C_VEL
LIN {X 0,Y 396.721,Z 570.589,A -85,B 0,C 180,E1 15643.453,E2 15643.453} C_VEL
LIN {X 0,Y 399.538,Z 576.401,A -85,B 0,C 180,E1 15640.406,E2 15640.406} C_VEL
LIN {X 0,Y 401.883,Z 581.131,A -85,B 0,C 180,E1 15638.24,E2 15638.24} C_VEL
LIN {X 0,Y 405.6,Z 588.616,A -85,B 0,C 180,E1 15635.223,E2 15635.223} C_VEL
LIN {X 0,Y 410.853,Z 600.236,A -85,B 0,C 180,E1 15631.351,E2 15631.351} C_VEL
LIN {X 0,Y 415.143,Z 610.224,A -85,B 0,C 180,E1 15628.57,E2 15628.57} C_VEL
LIN {X 0,Y 423.141,Z 622.653,A -85,B 0,C 180,E1 15626.186,E2 15626.186} C_VEL
LIN {X 0,Y 431.598,Z 636.427,A -85,B 0,C 180,E1 15623.912,E2 15623.912} C_VEL
LIN {X 0,Y 440.547,Z 652.077,A -85,B 0,C 180,E1 15621.712,E2 15621.712} C_VEL
LIN {X 0,Y 443.32,Z 657.546,A -85,B 0,C 180,E1 15621.055,E2 15621.055} C_VEL
LIN {X 0,Y 448.806,Z 707.472,A -85,B 0,C 180,E1 15618.854,E2 15618.854} C_VEL
LIN {X 0,Y 449.894,Z 719.55,A -85,B 0,C 180,E1 15618.386,E2 15618.386} C_VEL
LIN {X 0,Y 438.797,Z 948.139,A -85,B 0,C 180,E1 15614.82,E2 15614.82} C_VEL
LIN {X 0,Y 436.445,Z 970.869,A -85,B 0,C 180,E1 15614.302,E2 15614.302} C_VEL
LIN {X 0,Y 433.299,Z 992.491,A -85,B 0,C 180,E1 15613.627,E2 15613.627} C_VEL
LIN {X 0,Y 429.386,Z 1013.405,A -85,B 0,C 180,E1 15612.748,E2 15612.748} C_VEL
LIN {X 0,Y 424.63,Z 1034.807,A -85,B 0,C 180,E1 15611.607,E2 15611.607} C_VEL
LIN {X 0,Y 419.815,Z 1053.52,A -85,B 0,C 180,E1 15610.377,E2 15610.377} C_VEL
LIN {X 0,Y 414.3,Z 1072.42,A -85,B 0,C 180,E1 15608.864,E2 15608.864} C_VEL
LIN {X 0,Y 408.473,Z 1090.714,A -85,B 0,C 180,E1 15607.112,E2 15607.112} C_VEL
LIN {X 0,Y 402.449,Z 1107.936,A -85,B 0,C 180,E1 15605.11,E2 15605.11} C_VEL
LIN {X 0,Y 396.4,Z 1124.297,A -85,B 0,C 180,E1 15602.841,E2 15602.841} C_VEL
LIN {X 0,Y 390.792,Z 1138.897,A -85,B 0,C 180,E1 15600.428,E2 15600.428} C_VEL
LIN {X 0,Y 385.594,Z 1152.015,A -85,B 0,C 180,E1 15597.823,E2 15597.823} C_VEL
LIN {X 0,Y 380.909,Z 1164.022,A -85,B 0,C 180,E1 15595,E2 15595} C_VEL
LIN {X 0,Y 376.848,Z 1174.594,A -85,B 0,C 180,E1 15591.969,E2 15591.969} C_VEL
LIN {X 0,Y 373.386,Z 1184.295,A -85,B 0,C 180,E1 15588.561,E2 15588.561} C_VEL
LIN {X 0,Y 370.94,Z 1192.064,A -85,B 0,C 180,E1 15585.157,E2 15585.157} C_VEL
LIN {X 0,Y 369.353,Z 1198.002,A -85,B 0,C 180,E1 15581.714,E2 15581.714} C_VEL
LIN {X 0,Y 368.45,Z 1202.543,A -85,B 0,C 180,E1 15578.112,E2 15578.112} C_VEL
LIN {X 0,Y 368.099,Z 1205.223,A -85,B 0,C 180,E1 15574.83,E2 15574.83} C_VEL
LIN {X 0,Y 367.992,Z 1206.549,A -85,B 0,C 180,E1 15571.401,E2 15571.401} C_VEL
LIN {X 0,Y 367.996,Z 1206.522,A -85,B 0,C 180,E1 15568.287,E2 15568.287} C_VEL
LIN {X 0,Y 368.121,Z 1204.977,A -85,B 0,C 180,E1 15564.701,E2 15564.701} C_VEL
LIN {X 0,Y 368.512,Z 1202.197,A -85,B 0,C 180,E1 15561.418,E2 15561.418} C_VEL
LIN {X 0,Y 369.436,Z 1197.687,A -85,B 0,C 180,E1 15557.972,E2 15557.972} C_VEL
LIN {X 0,Y 371.077,Z 1191.644,A -85,B 0,C 180,E1 15554.529,E2 15554.529} C_VEL
LIN {X 0,Y 373.603,Z 1183.737,A -85,B 0,C 180,E1 15551.106,E2 15551.106} C_VEL
LIN {X 0,Y 377.121,Z 1173.933,A -85,B 0,C 180,E1 15547.719,E2 15547.719} C_VEL
LIN {X 0,Y 381.251,Z 1163.262,A -85,B 0,C 180,E1 15544.692,E2 15544.692} C_VEL
LIN {X 0,Y 385.999,Z 1151.118,A -85,B 0,C 180,E1 15541.872,E2 15541.872} C_VEL
LIN {X 0,Y 391.767,Z 1136.494,A -85,B 0,C 180,E1 15539.044,E2 15539.044} C_VEL
LIN {X 0,Y 392.347,Z 1134.996,A -85,B 0,C 180,E1 15538.784,E2 15538.784} C_VEL
LIN {X 0,Y 393.353,Z 1130.312,A -85,B 0,C 180,E1 15537.902,E2 15537.902} C_VEL
LIN {X 0,Y 392.997,Z 1118.275,A -85,B 0,C 180,E1 15535.55,E2 15535.55} C_VEL
LIN {X 0,Y 394.215,Z 1113.033,A -85,B 0,C 180,E1 15534.73,E2 15534.73} C_VEL
LIN {X 0,Y 400.407,Z 1096.071,A -85,B 0,C 180,E1 15532.642,E2 15532.642} C_VEL
LIN {X 0,Y 406.529,Z 1078.188,A -85,B 0,C 180,E1 15530.796,E2 15530.796} C_VEL
LIN {X 0,Y 412.097,Z 1060.111,A -85,B 0,C 180,E1 15529.257,E2 15529.257} C_VEL
LIN {X 0,Y 417.73,Z 1039.767,A -85,B 0,C 180,E1 15527.826,E2 15527.826} C_VEL
LIN {X 0,Y 422.432,Z 1020.24,A -85,B 0,C 180,E1 15526.71,E2 15526.71} C_VEL
LIN {X 0,Y 426.677,Z 999.207,A -85,B 0,C 180,E1 15525.755,E2 15525.755} C_VEL
LIN {X 0,Y 430.278,Z 977.616,A -85,B 0,C 180,E1 15524.997,E2 15524.997} C_VEL
LIN {X 0,Y 432.935,Z 955.312,A -85,B 0,C 180,E1 15524.439,E2 15524.439} C_VEL
LIN {X 0,Y 434.835,Z 925.959,A -85,B 0,C 180,E1 15523.919,E2 15523.919} C_VEL
LIN {X 0,Y 445.009,Z 719.047,A -85,B 0,C 180,E1 15520.668,E2 15520.668} C_VEL
LIN {X 0,Y 439.518,Z 665.976,A -85,B 0,C 180,E1 15518.332,E2 15518.332} C_VEL
LIN {X 0,Y 438.88,Z 661.318,A -85,B 0,C 180,E1 15518.086,E2 15518.086} C_VEL
LIN {X 0,Y 429.994,Z 645.402,A -85,B 0,C 180,E1 15515.873,E2 15515.873} C_VEL
LIN {X 0,Y 421.29,Z 630.824,A -85,B 0,C 180,E1 15513.492,E2 15513.492} C_VEL
LIN {X 0,Y 413.382,Z 618.339,A -85,B 0,C 180,E1 15511.1,E2 15511.1} C_VEL
LIN {X 0,Y 406.051,Z 607.038,A -85,B 0,C 180,E1 15508.537,E2 15508.537} C_VEL
LIN {X 0,Y 401.758,Z 597.36,A -85,B 0,C 180,E1 15505.345,E2 15505.345} C_VEL
LIN {X 0,Y 398.248,Z 589.788,A -85,B 0,C 180,E1 15502.435,E2 15502.435} C_VEL
LIN {X 0,Y 395.986,Z 585.182,A -85,B 0,C 180,E1 15500.393,E2 15500.393} C_VEL
LIN {X 0,Y 393.944,Z 581.006,A -85,B 0,C 180,E1 15498.334,E2 15498.334} C_VEL
LIN {X 0,Y 391.895,Z 576.844,A -85,B 0,C 180,E1 15495.995,E2 15495.995} C_VEL
LIN {X 0,Y 389.498,Z 572.125,A -85,B 0,C 180,E1 15492.755,E2 15492.755} C_VEL
LIN {X 0,Y 387.114,Z 567.462,A -85,B 0,C 180,E1 15488.317,E2 15488.317} C_VEL
LIN {X 0,Y 385.278,Z 564.949,A -85,B 0,C 180,E1 15482.678,E2 15482.678} C_VEL
LIN {X 0,Y 385.188,Z 564.693,A -85,B 0,C 180,E1 15479.108,E2 15479.108} C_VEL
LIN {X 0,Y 386.006,Z 566.182,A -85,B 0,C 180,E1 15474.649,E2 15474.649} C_VEL
LIN {X 0,Y 387.539,Z 568.139,A -85,B 0,C 180,E1 15471.394,E2 15471.394} C_VEL
LIN {X 0,Y 390.149,Z 573.163,A -85,B 0,C 180,E1 15466.966,E2 15466.966} C_VEL
LIN {X 0,Y 391.981,Z 576.662,A -85,B 0,C 180,E1 15464.767,E2 15464.767} C_VEL
LIN {X 0,Y 394.386,Z 579.391,A -85,B 0,C 180,E1 15463.579,E2 15463.579} C_VEL
LIN {X 0,Y 399.373,Z 584.812,A -85,B 0,C 180,E1 15461.422,E2 15461.422} C_VEL
LIN {X 0,Y 404.454,Z 590.606,A -85,B 0,C 180,E1 15459.448,E2 15459.448} C_VEL
LIN {X 0,Y 411.882,Z 599.255,A -85,B 0,C 180,E1 15456.879,E2 15456.879} C_VEL
LIN {X 0,Y 422.813,Z 613.192,A -85,B 0,C 180,E1 15453.565,E2 15453.565} C_VEL
LIN {X 0,Y 432.892,Z 627.261,A -85,B 0,C 180,E1 15450.87,E2 15450.87} C_VEL
LIN {X 0,Y 443.283,Z 642.832,A -85,B 0,C 180,E1 15448.369,E2 15448.369} C_VEL
LIN {X 0,Y 451.045,Z 655.654,A -85,B 0,C 180,E1 15446.631,E2 15446.631} C_VEL
LIN {X 0,Y 436.61,Z 892.873,A -85,B 0,C 180,E1 15442.564,E2 15442.564} C_VEL
LIN {X 0,Y 434.008,Z 931.883,A -85,B 0,C 180,E1 15441.848,E2 15441.848} C_VEL
LIN {X 0,Y 431.328,Z 955.256,A -85,B 0,C 180,E1 15441.234,E2 15441.234} C_VEL
LIN {X 0,Y 427.698,Z 979.59,A -85,B 0,C 180,E1 15440.38,E2 15440.38} C_VEL
LIN {X 0,Y 423.825,Z 1000.582,A -85,B 0,C 180,E1 15439.432,E2 15439.432} C_VEL
LIN {X 0,Y 418.826,Z 1023.779,A -85,B 0,C 180,E1 15438.145,E2 15438.145} C_VEL
LIN {X 0,Y 413.743,Z 1044.148,A -85,B 0,C 180,E1 15436.77,E2 15436.77} C_VEL
LIN {X 0,Y 407.412,Z 1066.959,A -85,B 0,C 180,E1 15434.915,E2 15434.915} C_VEL
LIN {X 0,Y 401.72,Z 1085.746,A -85,B 0,C 180,E1 15433.095,E2 15433.095} C_VEL
LIN {X 0,Y 395.455,Z 1105.007,A -85,B 0,C 180,E1 15430.886,E2 15430.886} C_VEL
LIN {X 0,Y 389.783,Z 1121.715,A -85,B 0,C 180,E1 15428.646,E2 15428.646} C_VEL
LIN {X 0,Y 383.66,Z 1139.089,A -85,B 0,C 180,E1 15425.9,E2 15425.9} C_VEL
LIN {X 0,Y 378.345,Z 1154.253,A -85,B 0,C 180,E1 15423.094,E2 15423.094} C_VEL
LIN {X 0,Y 373.486,Z 1168.155,A -85,B 0,C 180,E1 15420.041,E2 15420.041} C_VEL
LIN {X 0,Y 369.225,Z 1181.118,A -85,B 0,C 180,E1 15416.713,E2 15416.713} C_VEL
LIN {X 0,Y 365.842,Z 1192.059,A -85,B 0,C 180,E1 15413.316,E2 15413.316} C_VEL
LIN {X 0,Y 363.297,Z 1201.674,A -85,B 0,C 180,E1 15409.787,E2 15409.787} C_VEL
LIN {X 0,Y 361.567,Z 1209.436,A -85,B 0,C 180,E1 15406.218,E2 15406.218} C_VEL
LIN {X 0,Y 360.547,Z 1215.714,A -85,B 0,C 180,E1 15402.655,E2 15402.655} C_VEL
LIN {X 0,Y 360.078,Z 1220.28,A -85,B 0,C 180,E1 15399.107,E2 15399.107} C_VEL
LIN {X 0,Y 359.961,Z 1223.064,A -85,B 0,C 180,E1 15396.041,E2 15396.041} C_VEL
LIN {X 0,Y 359.943,Z 1224.953,A -85,B 0,C 180,E1 15392.547,E2 15392.547} C_VEL
LIN {X 0,Y 359.954,Z 1225.232,A -85,B 0,C 180,E1 15389.204,E2 15389.204} C_VEL
LIN {X 0,Y 359.953,Z 1224.371,A -85,B 0,C 180,E1 15386.177,E2 15386.177} C_VEL
LIN {X 0,Y 359.982,Z 1222.192,A -85,B 0,C 180,E1 15382.82,E2 15382.82} C_VEL
LIN {X 0,Y 360.249,Z 1218.137,A -85,B 0,C 180,E1 15379.121,E2 15379.121} C_VEL
LIN {X 0,Y 360.9,Z 1213.228,A -85,B 0,C 180,E1 15375.859,E2 15375.859} C_VEL
LIN {X 0,Y 362.329,Z 1205.709,A -85,B 0,C 180,E1 15371.997,E2 15371.997} C_VEL
LIN {X 0,Y 364.234,Z 1197.833,A -85,B 0,C 180,E1 15368.755,E2 15368.755} C_VEL
LIN {X 0,Y 367.202,Z 1187.502,A -85,B 0,C 180,E1 15365.208,E2 15365.208} C_VEL
LIN {X 0,Y 370.725,Z 1176.298,A -85,B 0,C 180,E1 15362.012,E2 15362.012} C_VEL
LIN {X 0,Y 375.353,Z 1162.657,A -85,B 0,C 180,E1 15358.706,E2 15358.706} C_VEL
LIN {X 0,Y 380.093,Z 1149.071,A -85,B 0,C 180,E1 15355.923,E2 15355.923} C_VEL
LIN {X 0,Y 386.04,Z 1132.219,A -85,B 0,C 180,E1 15352.974,E2 15352.974} C_VEL
LIN {X 0,Y 391.549,Z 1116.323,A -85,B 0,C 180,E1 15350.612,E2 15350.612} C_VEL
LIN {X 0,Y 398.22,Z 1096.381,A -85,B 0,C 180,E1 15348.097,E2 15348.097} C_VEL
LIN {X 0,Y 404.031,Z 1078.036,A -85,B 0,C 180,E1 15346.139,E2 15346.139} C_VEL
LIN {X 0,Y 410.024,Z 1057.589,A -85,B 0,C 180,E1 15344.299,E2 15344.299} C_VEL
LIN {X 0,Y 415.163,Z 1038.389,A -85,B 0,C 180,E1 15342.833,E2 15342.833} C_VEL
LIN {X 0,Y 420.563,Z 1015.678,A -85,B 0,C 180,E1 15341.393,E2 15341.393} C_VEL
LIN {X 0,Y 424.837,Z 995.004,A -85,B 0,C 180,E1 15340.312,E2 15340.312} C_VEL
LIN {X 0,Y 428.964,Z 971.12,A -85,B 0,C 180,E1 15339.315,E2 15339.315} C_VEL
LIN {X 0,Y 432.033,Z 949.099,A -85,B 0,C 180,E1 15338.6,E2 15338.6} C_VEL
LIN {X 0,Y 434.505,Z 924.339,A -85,B 0,C 180,E1 15338.015,E2 15338.015} C_VEL
LIN {X 0,Y 448.454,Z 695.376,A -85,B 0,C 180,E1 15334.052,E2 15334.052} C_VEL
LIN {X 0,Y 450.811,Z 655.196,A -85,B 0,C 180,E1 15333.352,E2 15333.352} C_VEL
LIN {X 0,Y 440.828,Z 639.083,A -85,B 0,C 180,E1 15331.104,E2 15331.104} C_VEL
LIN {X 0,Y 429.657,Z 622.606,A -85,B 0,C 180,E1 15328.343,E2 15328.343} C_VEL
LIN {X 0,Y 419.12,Z 608.412,A -85,B 0,C 180,E1 15325.431,E2 15325.431} C_VEL
LIN {X 0,Y 409.832,Z 596.94,A -85,B 0,C 180,E1 15322.522,E2 15322.522} C_VEL
LIN {X 0,Y 402.497,Z 588.205,A -85,B 0,C 180,E1 15319.898,E2 15319.898} C_VEL
LIN {X 0,Y 396.637,Z 581.786,A -85,B 0,C 180,E1 15317.533,E2 15317.533} C_VEL
LIN {X 0,Y 391.972,Z 576.674,A -85,B 0,C 180,E1 15315.385,E2 15315.385} C_VEL
LIN {X 0,Y 389.711,Z 572.3,A -85,B 0,C 180,E1 15312.597,E2 15312.597} C_VEL
LIN {X 0,Y 387.171,Z 567.488,A -85,B 0,C 180,E1 15308.166,E2 15308.166} C_VEL
LIN {X 0,Y 385.151,Z 564.69,A -85,B 0,C 180,E1 15302.381,E2 15302.381} C_VEL
LIN {X 0,Y 385.017,Z 564.332,A -85,B 0,C 180,E1 15298.661,E2 15298.661} C_VEL
LIN {X 0,Y 385.732,Z 565.862,A -85,B 0,C 180,E1 15294.198,E2 15294.198} C_VEL
LIN {X 0,Y 387.322,Z 567.87,A -85,B 0,C 180,E1 15290.79,E2 15290.79} C_VEL
LIN {X 0,Y 389.993,Z 573.134,A -85,B 0,C 180,E1 15286.205,E2 15286.205} C_VEL
LIN {X 0,Y 392.413,Z 577.968,A -85,B 0,C 180,E1 15283.113,E2 15283.113} C_VEL
LIN {X 0,Y 394.738,Z 582.627,A -85,B 0,C 180,E1 15280.62,E2 15280.62} C_VEL
LIN {X 0,Y 397.17,Z 587.725,A -85,B 0,C 180,E1 15278.279,E2 15278.279} C_VEL
LIN {X 0,Y 400.494,Z 594.472,A -85,B 0,C 180,E1 15275.516,E2 15275.516} C_VEL
LIN {X 0,Y 404.981,Z 604.752,A -85,B 0,C 180,E1 15272.023,E2 15272.023} C_VEL
LIN {X 0,Y 407.026,Z 608.89,A -85,B 0,C 180,E1 15270.855,E2 15270.855} C_VEL
LIN {X 0,Y 415.492,Z 621.738,A -85,B 0,C 180,E1 15268.073,E2 15268.073} C_VEL
LIN {X 0,Y 423.564,Z 634.648,A -85,B 0,C 180,E1 15265.711,E2 15265.711} C_VEL
LIN {X 0,Y 432.583,Z 650.087,A -85,B 0,C 180,E1 15263.316,E2 15263.316} C_VEL
LIN {X 0,Y 438.901,Z 661.737,A -85,B 0,C 180,E1 15261.76,E2 15261.76} C_VEL
LIN {X 0,Y 444.175,Z 712.029,A -85,B 0,C 180,E1 15259.52,E2 15259.52} C_VEL
LIN {X 0,Y 444.905,Z 720.989,A -85,B 0,C 180,E1 15259.174,E2 15259.174} C_VEL
LIN {X 0,Y 433.48,Z 947.797,A -85,B 0,C 180,E1 15255.611,E2 15255.611} C_VEL
LIN {X 0,Y 431.071,Z 970.546,A -85,B 0,C 180,E1 15255.092,E2 15255.092} C_VEL
LIN {X 0,Y 427.861,Z 992.103,A -85,B 0,C 180,E1 15254.418,E2 15254.418} C_VEL
LIN {X 0,Y 423.843,Z 1013.043,A -85,B 0,C 180,E1 15253.538,E2 15253.538} C_VEL
LIN {X 0,Y 418.864,Z 1034.85,A -85,B 0,C 180,E1 15252.37,E2 15252.37} C_VEL
LIN {X 0,Y 414.001,Z 1053.231,A -85,B 0,C 180,E1 15251.156,E2 15251.156} C_VEL
LIN {X 0,Y 408.434,Z 1071.836,A -85,B 0,C 180,E1 15249.664,E2 15249.664} C_VEL
LIN {X 0,Y 402.633,Z 1089.554,A -85,B 0,C 180,E1 15247.968,E2 15247.968} C_VEL
LIN {X 0,Y 396.482,Z 1106.673,A -85,B 0,C 180,E1 15245.986,E2 15245.986} C_VEL
LIN {X 0,Y 390.368,Z 1122.81,A -85,B 0,C 180,E1 15243.766,E2 15243.766} C_VEL
LIN {X 0,Y 384.825,Z 1136.688,A -85,B 0,C 180,E1 15241.483,E2 15241.483} C_VEL
LIN {X 0,Y 379.005,Z 1150.923,A -85,B 0,C 180,E1 15238.694,E2 15238.694} C_VEL
LIN {X 0,Y 374.049,Z 1163.107,A -85,B 0,C 180,E1 15235.83,E2 15235.83} C_VEL
LIN {X 0,Y 369.698,Z 1173.879,A -85,B 0,C 180,E1 15232.739,E2 15232.739} C_VEL
LIN {X 0,Y 366.151,Z 1183.307,A -85,B 0,C 180,E1 15229.46,E2 15229.46} C_VEL
LIN {X 0,Y 363.527,Z 1190.955,A -85,B 0,C 180,E1 15226.129,E2 15226.129} C_VEL
LIN {X 0,Y 361.627,Z 1197.49,A -85,B 0,C 180,E1 15222.454,E2 15222.454} C_VEL
LIN {X 0,Y 360.604,Z 1202.146,A -85,B 0,C 180,E1 15218.933,E2 15218.933} C_VEL
LIN {X 0,Y 360.14,Z 1205.107,A -85,B 0,C 180,E1 15215.416,E2 15215.416} C_VEL
LIN {X 0,Y 360.006,Z 1206.69,A -85,B 0,C 180,E1 15211.91,E2 15211.91} C_VEL
LIN {X 0,Y 359.992,Z 1206.79,A -85,B 0,C 180,E1 15208.727,E2 15208.727} C_VEL
LIN {X 0,Y 360.097,Z 1205.612,A -85,B 0,C 180,E1 15205.222,E2 15205.222} C_VEL
LIN {X 0,Y 360.443,Z 1203.007,A -85,B 0,C 180,E1 15201.867,E2 15201.867} C_VEL
LIN {X 0,Y 361.362,Z 1198.624,A -85,B 0,C 180,E1 15198.185,E2 15198.185} C_VEL
LIN {X 0,Y 362.981,Z 1192.768,A -85,B 0,C 180,E1 15194.666,E2 15194.666} C_VEL
LIN {X 0,Y 365.511,Z 1185.124,A -85,B 0,C 180,E1 15191.168,E2 15191.168} C_VEL
LIN {X 0,Y 368.873,Z 1176.154,A -85,B 0,C 180,E1 15187.866,E2 15187.866} C_VEL
LIN {X 0,Y 372.987,Z 1165.743,A -85,B 0,C 180,E1 15184.772,E2 15184.772} C_VEL
LIN {X 0,Y 378.059,Z 1153.359,A -85,B 0,C 180,E1 15181.73,E2 15181.73} C_VEL
LIN {X 0,Y 383.707,Z 1139.698,A -85,B 0,C 180,E1 15178.939,E2 15178.939} C_VEL
LIN {X 0,Y 389.472,Z 1125.212,A -85,B 0,C 180,E1 15176.499,E2 15176.499} C_VEL
LIN {X 0,Y 394.215,Z 1113.033,A -85,B 0,C 180,E1 15174.73,E2 15174.73} C_VEL
LIN {X 0,Y 395.484,Z 1107.736,A -85,B 0,C 180,E1 15173.925,E2 15173.925} C_VEL
LIN {X 0,Y 395.711,Z 1094.268,A -85,B 0,C 180,E1 15171.759,E2 15171.759} C_VEL
LIN {X 0,Y 396.968,Z 1088.409,A -85,B 0,C 180,E1 15171.048,E2 15171.048} C_VEL
LIN {X 0,Y 402.939,Z 1070.697,A -85,B 0,C 180,E1 15169.355,E2 15169.355} C_VEL
LIN {X 0,Y 409.045,Z 1050.524,A -85,B 0,C 180,E1 15167.763,E2 15167.763} C_VEL
LIN {X 0,Y 414.422,Z 1030.566,A -85,B 0,C 180,E1 15166.474,E2 15166.474} C_VEL
LIN {X 0,Y 419.155,Z 1009.573,A -85,B 0,C 180,E1 15165.401,E2 15165.401} C_VEL
LIN {X 0,Y 423.484,Z 986.404,A -85,B 0,C 180,E1 15164.482,E2 15164.482} C_VEL
LIN {X 0,Y 426.724,Z 964.24,A -85,B 0,C 180,E1 15163.835,E2 15163.835} C_VEL
LIN {X 0,Y 428.777,Z 941.523,A -85,B 0,C 180,E1 15163.368,E2 15163.368} C_VEL
LIN {X 0,Y 440.123,Z 720.559,A -85,B 0,C 180,E1 15159.863,E2 15159.863} C_VEL
LIN {X 0,Y 434.94,Z 668.117,A -85,B 0,C 180,E1 15157.516,E2 15157.516} C_VEL
LIN {X 0,Y 434.514,Z 665.785,A -85,B 0,C 180,E1 15157.368,E2 15157.368} C_VEL
LIN {X 0,Y 425.546,Z 649.572,A -85,B 0,C 180,E1 15155.044,E2 15155.044} C_VEL
LIN {X 0,Y 417.122,Z 635.348,A -85,B 0,C 180,E1 15152.64,E2 15152.64} C_VEL
LIN {X 0,Y 408.862,Z 622.17,A -85,B 0,C 180,E1 15150.008,E2 15150.008} C_VEL
LIN {X 0,Y 401.733,Z 611.584,A -85,B 0,C 180,E1 15147.457,E2 15147.457} C_VEL
LIN {X 0,Y 397.226,Z 604.368,A -85,B 0,C 180,E1 15145.496,E2 15145.496} C_VEL
LIN {X 0,Y 393.377,Z 596.014,A -85,B 0,C 180,E1 15142.255,E2 15142.255} C_VEL
LIN {X 0,Y 390.996,Z 591.128,A -85,B 0,C 180,E1 15140.04,E2 15140.04} C_VEL
LIN {X 0,Y 389.165,Z 587.286,A -85,B 0,C 180,E1 15138.113,E2 15138.113} C_VEL
LIN {X 0,Y 387.144,Z 583.162,A -85,B 0,C 180,E1 15135.735,E2 15135.735} C_VEL
LIN {X 0,Y 384.935,Z 578.656,A -85,B 0,C 180,E1 15132.603,E2 15132.603} C_VEL
LIN {X 0,Y 382.617,Z 574.052,A -85,B 0,C 180,E1 15128.113,E2 15128.113} C_VEL
LIN {X 0,Y 380.914,Z 571.636,A -85,B 0,C 180,E1 15122.558,E2 15122.558} C_VEL
LIN {X 0,Y 380.853,Z 571.429,A -85,B 0,C 180,E1 15118.947,E2 15118.947} C_VEL
LIN {X 0,Y 381.719,Z 573.008,A -85,B 0,C 180,E1 15114.438,E2 15114.438} C_VEL
LIN {X 0,Y 383.115,Z 574.831,A -85,B 0,C 180,E1 15111.445,E2 15111.445} C_VEL
LIN {X 0,Y 385.234,Z 578.85,A -85,B 0,C 180,E1 15107.864,E2 15107.864} C_VEL
LIN {X 0,Y 387.104,Z 581.117,A -85,B 0,C 180,E1 15106.71,E2 15106.71} C_VEL
LIN {X 0,Y 392.064,Z 586.157,A -85,B 0,C 180,E1 15104.164,E2 15104.164} C_VEL
LIN {X 0,Y 397.783,Z 592.651,A -85,B 0,C 180,E1 15101.611,E2 15101.611} C_VEL
LIN {X 0,Y 402.553,Z 598.161,A -85,B 0,C 180,E1 15099.727,E2 15099.727} C_VEL
LIN {X 0,Y 409.497,Z 606.373,A -85,B 0,C 180,E1 15097.269,E2 15097.269} C_VEL
LIN {X 0,Y 420.051,Z 620.042,A -85,B 0,C 180,E1 15093.986,E2 15093.986} C_VEL
LIN {X 0,Y 429.874,Z 633.961,A -85,B 0,C 180,E1 15091.293,E2 15091.293} C_VEL
LIN {X 0,Y 439.879,Z 649.184,A -85,B 0,C 180,E1 15088.822,E2 15088.822} C_VEL
LIN {X 0,Y 446.053,Z 659.516,A -85,B 0,C 180,E1 15087.392,E2 15087.392} C_VEL
LIN {X 0,Y 431.127,Z 898.3,A -85,B 0,C 180,E1 15083.279,E2 15083.279} C_VEL
LIN {X 0,Y 428.646,Z 933.204,A -85,B 0,C 180,E1 15082.625,E2 15082.625} C_VEL
LIN {X 0,Y 425.946,Z 956.052,A -85,B 0,C 180,E1 15082.018,E2 15082.018} C_VEL
LIN {X 0,Y 422.108,Z 980.843,A -85,B 0,C 180,E1 15081.136,E2 15081.136} C_VEL
LIN {X 0,Y 418.024,Z 1002.253,A -85,B 0,C 180,E1 15080.156,E2 15080.156} C_VEL
LIN {X 0,Y 412.631,Z 1026.138,A -85,B 0,C 180,E1 15078.797,E2 15078.797} C_VEL
LIN {X 0,Y 407.431,Z 1046.275,A -85,B 0,C 180,E1 15077.41,E2 15077.41} C_VEL
LIN {X 0,Y 401.296,Z 1067.509,A -85,B 0,C 180,E1 15075.65,E2 15075.65} C_VEL
LIN {X 0,Y 395.237,Z 1086.861,A -85,B 0,C 180,E1 15073.75,E2 15073.75} C_VEL
LIN {X 0,Y 388.88,Z 1105.635,A -85,B 0,C 180,E1 15071.556,E2 15071.556} C_VEL
LIN {X 0,Y 382.815,Z 1122.875,A -85,B 0,C 180,E1 15069.203,E2 15069.203} C_VEL
LIN {X 0,Y 376.642,Z 1139.648,A -85,B 0,C 180,E1 15066.487,E2 15066.487} C_VEL
LIN {X 0,Y 370.958,Z 1155.213,A -85,B 0,C 180,E1 15063.542,E2 15063.542} C_VEL
LIN {X 0,Y 365.845,Z 1169.202,A -85,B 0,C 180,E1 15060.372,E2 15060.372} C_VEL
LIN {X 0,Y 361.451,Z 1181.949,A -85,B 0,C 180,E1 15056.979,E2 15056.979} C_VEL
LIN {X 0,Y 358.11,Z 1192.293,A -85,B 0,C 180,E1 15053.677,E2 15053.677} C_VEL
LIN {X 0,Y 355.406,Z 1201.97,A -85,B 0,C 180,E1 15050.003,E2 15050.003} C_VEL
LIN {X 0,Y 353.636,Z 1209.533,A -85,B 0,C 180,E1 15046.424,E2 15046.424} C_VEL
LIN {X 0,Y 352.546,Z 1215.909,A -85,B 0,C 180,E1 15042.668,E2 15042.668} C_VEL
LIN {X 0,Y 352.081,Z 1220.239,A -85,B 0,C 180,E1 15039.151,E2 15039.151} C_VEL
LIN {X 0,Y 351.955,Z 1223.085,A -85,B 0,C 180,E1 15035.87,E2 15035.87} C_VEL
LIN {X 0,Y 351.954,Z 1224.811,A -85,B 0,C 180,E1 15032.279,E2 15032.279} C_VEL
LIN {X 0,Y 351.961,Z 1225.004,A -85,B 0,C 180,E1 15029.023,E2 15029.023} C_VEL
LIN {X 0,Y 351.956,Z 1224.093,A -85,B 0,C 180,E1 15025.927,E2 15025.927} C_VEL
LIN {X 0,Y 351.98,Z 1221.735,A -85,B 0,C 180,E1 15022.327,E2 15022.327} C_VEL
LIN {X 0,Y 352.308,Z 1217.705,A -85,B 0,C 180,E1 15018.707,E2 15018.707} C_VEL
LIN {X 0,Y 353.021,Z 1212.791,A -85,B 0,C 180,E1 15015.4,E2 15015.4} C_VEL
LIN {X 0,Y 354.602,Z 1205.109,A -85,B 0,C 180,E1 15011.42,E2 15011.42} C_VEL
LIN {X 0,Y 356.669,Z 1197.173,A -85,B 0,C 180,E1 15008.109,E2 15008.109} C_VEL
LIN {X 0,Y 360.02,Z 1186.177,A -85,B 0,C 180,E1 15004.326,E2 15004.326} C_VEL
LIN {X 0,Y 363.622,Z 1175.44,A -85,B 0,C 180,E1 15001.236,E2 15001.236} C_VEL
LIN {X 0,Y 368.787,Z 1160.919,A -85,B 0,C 180,E1 14997.717,E2 14997.717} C_VEL
LIN {X 0,Y 373.847,Z 1147.179,A -85,B 0,C 180,E1 14994.899,E2 14994.899} C_VEL
LIN {X 0,Y 379.949,Z 1130.449,A -85,B 0,C 180,E1 14991.991,E2 14991.991} C_VEL
LIN {X 0,Y 385.941,Z 1113.88,A -85,B 0,C 180,E1 14989.536,E2 14989.536} C_VEL
LIN {X 0,Y 392.278,Z 1095.444,A -85,B 0,C 180,E1 14987.231,E2 14987.231} C_VEL
LIN {X 0,Y 398.585,Z 1076.214,A -85,B 0,C 180,E1 14985.179,E2 14985.179} C_VEL
LIN {X 0,Y 404.554,Z 1056.2,A -85,B 0,C 180,E1 14983.396,E2 14983.396} C_VEL
LIN {X 0,Y 410.053,Z 1036.193,A -85,B 0,C 180,E1 14981.878,E2 14981.878} C_VEL
LIN {X 0,Y 415.159,Z 1014.981,A -85,B 0,C 180,E1 14980.55,E2 14980.55} C_VEL
LIN {X 0,Y 419.594,Z 994.071,A -85,B 0,C 180,E1 14979.46,E2 14979.46} C_VEL
LIN {X 0,Y 423.67,Z 970.864,A -85,B 0,C 180,E1 14978.498,E2 14978.498} C_VEL
LIN {X 0,Y 426.817,Z 948.789,A -85,B 0,C 180,E1 14977.784,E2 14977.784} C_VEL
LIN {X 0,Y 429.298,Z 924.238,A -85,B 0,C 180,E1 14977.205,E2 14977.205} C_VEL
LIN {X 0,Y 443.913,Z 690.948,A -85,B 0,C 180,E1 14973.154,E2 14973.154} C_VEL
LIN {X 0,Y 445.802,Z 659.039,A -85,B 0,C 180,E1 14972.589,E2 14972.589} C_VEL
LIN {X 0,Y 436.367,Z 643.838,A -85,B 0,C 180,E1 14970.386,E2 14970.386} C_VEL
LIN {X 0,Y 426.337,Z 628.848,A -85,B 0,C 180,E1 14967.821,E2 14967.821} C_VEL
LIN {X 0,Y 416.416,Z 615.276,A -85,B 0,C 180,E1 14965,E2 14965} C_VEL
LIN {X 0,Y 407.381,Z 603.942,A -85,B 0,C 180,E1 14962.095,E2 14962.095} C_VEL
LIN {X 0,Y 400.099,Z 595.164,A -85,B 0,C 180,E1 14959.413,E2 14959.413} C_VEL
LIN {X 0,Y 394.526,Z 589.005,A -85,B 0,C 180,E1 14957.097,E2 14957.097} C_VEL
LIN {X 0,Y 390.248,Z 584.208,A -85,B 0,C 180,E1 14955.074,E2 14955.074} C_VEL
LIN {X 0,Y 386.008,Z 579.582,A -85,B 0,C 180,E1 14952.796,E2 14952.796} C_VEL
LIN {X 0,Y 384.317,Z 577.796,A -85,B 0,C 180,E1 14951.404,E2 14951.404} C_VEL
LIN {X 0,Y 382.751,Z 574.142,A -85,B 0,C 180,E1 14948.087,E2 14948.087} C_VEL
LIN {X 0,Y 380.812,Z 571.419,A -85,B 0,C 180,E1 14942.408,E2 14942.408} C_VEL
LIN {X 0,Y 380.669,Z 571.027,A -85,B 0,C 180,E1 14938.796,E2 14938.796} C_VEL
LIN {X 0,Y 381.34,Z 572.531,A -85,B 0,C 180,E1 14934.282,E2 14934.282} C_VEL
LIN {X 0,Y 382.902,Z 574.632,A -85,B 0,C 180,E1 14930.771,E2 14930.771} C_VEL
LIN {X 0,Y 385.426,Z 579.646,A -85,B 0,C 180,E1 14926.345,E2 14926.345} C_VEL
LIN {X 0,Y 387.786,Z 584.498,A -85,B 0,C 180,E1 14923.215,E2 14923.215} C_VEL
LIN {X 0,Y 390.066,Z 589.186,A -85,B 0,C 180,E1 14920.69,E2 14920.69} C_VEL
LIN {X 0,Y 392.317,Z 593.952,A -85,B 0,C 180,E1 14918.469,E2 14918.469} C_VEL
LIN {X 0,Y 395.574,Z 600.716,A -85,B 0,C 180,E1 14915.668,E2 14915.668} C_VEL
LIN {X 0,Y 398.171,Z 606.323,A -85,B 0,C 180,E1 14913.77,E2 14913.77} C_VEL
LIN {X 0,Y 405.788,Z 617.656,A -85,B 0,C 180,E1 14910.879,E2 14910.879} C_VEL
LIN {X 0,Y 413.815,Z 630.082,A -85,B 0,C 180,E1 14908.214,E2 14908.214} C_VEL
LIN {X 0,Y 421.531,Z 642.86,A -85,B 0,C 180,E1 14905.917,E2 14905.917} C_VEL
LIN {X 0,Y 430.39,Z 658.338,A -85,B 0,C 180,E1 14903.526,E2 14903.526} C_VEL
LIN {X 0,Y 434.605,Z 666.46,A -85,B 0,C 180,E1 14902.454,E2 14902.454} C_VEL
LIN {X 0,Y 439.74,Z 718.04,A -85,B 0,C 180,E1 14900.138,E2 14900.138} C_VEL
LIN {X 0,Y 439.984,Z 722.752,A -85,B 0,C 180,E1 14899.975,E2 14899.975} C_VEL
LIN {X 0,Y 428.241,Z 947.566,A -85,B 0,C 180,E1 14896.42,E2 14896.42} C_VEL
LIN {X 0,Y 425.764,Z 970.351,A -85,B 0,C 180,E1 14895.897,E2 14895.897} C_VEL
LIN {X 0,Y 422.506,Z 991.716,A -85,B 0,C 180,E1 14895.231,E2 14895.231} C_VEL
LIN {X 0,Y 418.382,Z 1012.681,A -85,B 0,C 180,E1 14894.348,E2 14894.348} C_VEL
LIN {X 0,Y 413.36,Z 1034.182,A -85,B 0,C 180,E1 14893.199,E2 14893.199} C_VEL
LIN {X 0,Y 408.266,Z 1052.942,A -85,B 0,C 180,E1 14891.958,E2 14891.958} C_VEL
LIN {X 0,Y 402.28,Z 1072.375,A -85,B 0,C 180,E1 14890.386,E2 14890.386} C_VEL
LIN {X 0,Y 396.282,Z 1090.139,A -85,B 0,C 180,E1 14888.666,E2 14888.666} C_VEL
LIN {X 0,Y 389.996,Z 1107.034,A -85,B 0,C 180,E1 14886.681,E2 14886.681} C_VEL
LIN {X 0,Y 383.683,Z 1123.122,A -85,B 0,C 180,E1 14884.436,E2 14884.436} C_VEL
LIN {X 0,Y 377.615,Z 1137.807,A -85,B 0,C 180,E1 14881.976,E2 14881.976} C_VEL
LIN {X 0,Y 371.623,Z 1151.872,A -85,B 0,C 180,E1 14879.142,E2 14879.142} C_VEL
LIN {X 0,Y 366.517,Z 1163.956,A -85,B 0,C 180,E1 14876.227,E2 14876.227} C_VEL
LIN {X 0,Y 362.041,Z 1174.572,A -85,B 0,C 180,E1 14873.089,E2 14873.089} C_VEL
LIN {X 0,Y 358.205,Z 1184.306,A -85,B 0,C 180,E1 14869.57,E2 14869.57} C_VEL
LIN {X 0,Y 355.434,Z 1192.188,A -85,B 0,C 180,E1 14866.002,E2 14866.002} C_VEL
LIN {X 0,Y 353.608,Z 1198.186,A -85,B 0,C 180,E1 14862.409,E2 14862.409} C_VEL
LIN {X 0,Y 352.549,Z 1202.808,A -85,B 0,C 180,E1 14858.645,E2 14858.645} C_VEL
LIN {X 0,Y 352.129,Z 1205.529,A -85,B 0,C 180,E1 14855.213,E2 14855.213} C_VEL
LIN {X 0,Y 351.998,Z 1206.958,A -85,B 0,C 180,E1 14851.465,E2 14851.465} C_VEL
LIN {X 0,Y 352.002,Z 1206.93,A -85,B 0,C 180,E1 14848.209,E2 14848.209} C_VEL
LIN {X 0,Y 352.147,Z 1205.388,A -85,B 0,C 180,E1 14844.46,E2 14844.46} C_VEL
LIN {X 0,Y 352.596,Z 1202.61,A -85,B 0,C 180,E1 14841.027,E2 14841.027} C_VEL
LIN {X 0,Y 353.646,Z 1198.109,A -85,B 0,C 180,E1 14837.426,E2 14837.426} C_VEL
LIN {X 0,Y 355.487,Z 1192.082,A -85,B 0,C 180,E1 14833.832,E2 14833.832} C_VEL
LIN {X 0,Y 358.281,Z 1184.181,A -85,B 0,C 180,E1 14830.265,E2 14830.265} C_VEL
LIN {X 0,Y 362.145,Z 1174.406,A -85,B 0,C 180,E1 14826.746,E2 14826.746} C_VEL
LIN {X 0,Y 366.648,Z 1163.76,A -85,B 0,C 180,E1 14823.608,E2 14823.608} C_VEL
LIN {X 0,Y 371.779,Z 1151.64,A -85,B 0,C 180,E1 14820.694,E2 14820.694} C_VEL
LIN {X 0,Y 377.799,Z 1137.525,A -85,B 0,C 180,E1 14817.863,E2 14817.863} C_VEL
LIN {X 0,Y 383.511,Z 1123.713,A -85,B 0,C 180,E1 14815.546,E2 14815.546} C_VEL
LIN {X 0,Y 390.103,Z 1106.985,A -85,B 0,C 180,E1 14813.203,E2 14813.203} C_VEL
LIN {X 0,Y 396.484,Z 1089.84,A -85,B 0,C 180,E1 14811.194,E2 14811.194} C_VEL
LIN {X 0,Y 396.968,Z 1088.409,A -85,B 0,C 180,E1 14811.048,E2 14811.048} C_VEL
LIN {X 0,Y 398.25,Z 1082.521,A -85,B 0,C 180,E1 14810.354,E2 14810.354} C_VEL
LIN {X 0,Y 398.779,Z 1067.729,A -85,B 0,C 180,E1 14808.393,E2 14808.393} C_VEL
LIN {X 0,Y 400.054,Z 1061.338,A -85,B 0,C 180,E1 14807.776,E2 14807.776} C_VEL
LIN {X 0,Y 405.788,Z 1042.1,A -85,B 0,C 180,E1 14806.377,E2 14806.377} C_VEL
LIN {X 0,Y 410.873,Z 1022.234,A -85,B 0,C 180,E1 14805.211,E2 14805.211} C_VEL
LIN {X 0,Y 415.729,Z 999.861,A -85,B 0,C 180,E1 14804.167,E2 14804.167} C_VEL
LIN {X 0,Y 419.391,Z 979.16,A -85,B 0,C 180,E1 14803.427,E2 14803.427} C_VEL
LIN {X 0,Y 422.318,Z 956.717,A -85,B 0,C 180,E1 14802.845,E2 14802.845} C_VEL
LIN {X 0,Y 424.167,Z 932.919,A -85,B 0,C 180,E1 14802.394,E2 14802.394} C_VEL
LIN {X 0,Y 435.318,Z 721.965,A -85,B 0,C 180,E1 14799.035,E2 14799.035} C_VEL
LIN {X 0,Y 430.51,Z 670.943,A -85,B 0,C 180,E1 14796.717,E2 14796.717} C_VEL
LIN {X 0,Y 423.054,Z 657.092,A -85,B 0,C 180,E1 14794.723,E2 14794.723} C_VEL
LIN {X 0,Y 414.482,Z 642.293,A -85,B 0,C 180,E1 14792.218,E2 14792.218} C_VEL
LIN {X 0,Y 406.659,Z 629.512,A -85,B 0,C 180,E1 14789.659,E2 14789.659} C_VEL
LIN {X 0,Y 399.471,Z 618.625,A -85,B 0,C 180,E1 14787.02,E2 14787.02} C_VEL
LIN {X 0,Y 393.885,Z 610.264,A -85,B 0,C 180,E1 14784.683,E2 14784.683} C_VEL
LIN {X 0,Y 388.363,Z 601.943,A -85,B 0,C 180,E1 14781.921,E2 14781.921} C_VEL
LIN {X 0,Y 386.18,Z 597.361,A -85,B 0,C 180,E1 14779.827,E2 14779.827} C_VEL
LIN {X 0,Y 384.385,Z 593.549,A -85,B 0,C 180,E1 14777.876,E2 14777.876} C_VEL
LIN {X 0,Y 382.548,Z 589.665,A -85,B 0,C 180,E1 14775.618,E2 14775.618} C_VEL
LIN {X 0,Y 380.502,Z 585.322,A -85,B 0,C 180,E1 14772.598,E2 14772.598} C_VEL
LIN {X 0,Y 378.204,Z 580.717,A -85,B 0,C 180,E1 14768.055,E2 14768.055} C_VEL
LIN {X 0,Y 376.568,Z 578.361,A -85,B 0,C 180,E1 14762.587,E2 14762.587} C_VEL
LIN {X 0,Y 376.51,Z 578.15,A -85,B 0,C 180,E1 14758.935,E2 14758.935} C_VEL
LIN {X 0,Y 377.383,Z 579.756,A -85,B 0,C 180,E1 14754.374,E2 14754.374} C_VEL
LIN {X 0,Y 378.768,Z 581.414,A -85,B 0,C 180,E1 14751.652,E2 14751.652} C_VEL
LIN {X 0,Y 382.499,Z 585.614,A -85,B 0,C 180,E1 14748.846,E2 14748.846} C_VEL
LIN {X 0,Y 384.877,Z 587.817,A -85,B 0,C 180,E1 14747.395,E2 14747.395} C_VEL
LIN {X 0,Y 390.477,Z 593.88,A -85,B 0,C 180,E1 14744.403,E2 14744.403} C_VEL
LIN {X 0,Y 395.798,Z 599.985,A -85,B 0,C 180,E1 14741.973,E2 14741.973} C_VEL
LIN {X 0,Y 400.489,Z 605.496,A -85,B 0,C 180,E1 14740.075,E2 14740.075} C_VEL
LIN {X 0,Y 407.224,Z 613.626,A -85,B 0,C 180,E1 14737.63,E2 14737.63} C_VEL
LIN {X 0,Y 417.316,Z 626.893,A -85,B 0,C 180,E1 14734.413,E2 14734.413} C_VEL
LIN {X 0,Y 426.868,Z 640.643,A -85,B 0,C 180,E1 14731.726,E2 14731.726} C_VEL
LIN {X 0,Y 436.614,Z 655.735,A -85,B 0,C 180,E1 14729.252,E2 14729.252} C_VEL
LIN {X 0,Y 441.131,Z 663.485,A -85,B 0,C 180,E1 14728.167,E2 14728.167} C_VEL
LIN {X 0,Y 425.726,Z 903.526,A -85,B 0,C 180,E1 14724.017,E2 14724.017} C_VEL
LIN {X 0,Y 423.243,Z 935.644,A -85,B 0,C 180,E1 14723.395,E2 14723.395} C_VEL
LIN {X 0,Y 420.498,Z 957.965,A -85,B 0,C 180,E1 14722.789,E2 14722.789} C_VEL
LIN {X 0,Y 416.508,Z 982.564,A -85,B 0,C 180,E1 14721.892,E2 14721.892} C_VEL
LIN {X 0,Y 412.293,Z 1003.933,A -85,B 0,C 180,E1 14720.899,E2 14720.899} C_VEL
LIN {X 0,Y 407.016,Z 1026.468,A -85,B 0,C 180,E1 14719.599,E2 14719.599} C_VEL
LIN {X 0,Y 401.666,Z 1046.577,A -85,B 0,C 180,E1 14718.205,E2 14718.205} C_VEL
LIN {X 0,Y 395.289,Z 1067.927,A -85,B 0,C 180,E1 14716.419,E2 14716.419} C_VEL
LIN {X 0,Y 388.996,Z 1087.383,A -85,B 0,C 180,E1 14714.489,E2 14714.489} C_VEL
LIN {X 0,Y 382.313,Z 1106.394,A -85,B 0,C 180,E1 14712.231,E2 14712.231} C_VEL
LIN {X 0,Y 375.768,Z 1124.309,A -85,B 0,C 180,E1 14709.735,E2 14709.735} C_VEL
LIN {X 0,Y 369.548,Z 1140.512,A -85,B 0,C 180,E1 14707.043,E2 14707.043} C_VEL
LIN {X 0,Y 363.765,Z 1155.659,A -85,B 0,C 180,E1 14704.106,E2 14704.106} C_VEL
LIN {X 0,Y 358.7,Z 1168.934,A -85,B 0,C 180,E1 14701.043,E2 14701.043} C_VEL
LIN {X 0,Y 354.07,Z 1181.702,A -85,B 0,C 180,E1 14697.588,E2 14697.588} C_VEL
LIN {X 0,Y 350.573,Z 1191.973,A -85,B 0,C 180,E1 14694.249,E2 14694.249} C_VEL
LIN {X 0,Y 347.718,Z 1201.594,A -85,B 0,C 180,E1 14690.537,E2 14690.537} C_VEL
LIN {X 0,Y 345.777,Z 1209.312,A -85,B 0,C 180,E1 14686.808,E2 14686.808} C_VEL
LIN {X 0,Y 344.632,Z 1215.541,A -85,B 0,C 180,E1 14683.079,E2 14683.079} C_VEL
LIN {X 0,Y 344.095,Z 1220.03,A -85,B 0,C 180,E1 14679.365,E2 14679.365} C_VEL
LIN {X 0,Y 343.961,Z 1222.878,A -85,B 0,C 180,E1 14676.007,E2 14676.007} C_VEL
LIN {X 0,Y 343.954,Z 1224.607,A -85,B 0,C 180,E1 14672.332,E2 14672.332} C_VEL
LIN {X 0,Y 343.964,Z 1224.799,A -85,B 0,C 180,E1 14669.001,E2 14669.001} C_VEL
LIN {X 0,Y 343.956,Z 1223.888,A -85,B 0,C 180,E1 14665.832,E2 14665.832} C_VEL
LIN {X 0,Y 343.99,Z 1221.526,A -85,B 0,C 180,E1 14662.148,E2 14662.148} C_VEL
LIN {X 0,Y 344.347,Z 1217.491,A -85,B 0,C 180,E1 14658.443,E2 14658.443} C_VEL
LIN {X 0,Y 345.113,Z 1212.572,A -85,B 0,C 180,E1 14655.058,E2 14655.058} C_VEL
LIN {X 0,Y 346.813,Z 1204.879,A -85,B 0,C 180,E1 14650.987,E2 14650.987} C_VEL
LIN {X 0,Y 349.02,Z 1196.938,A -85,B 0,C 180,E1 14647.604,E2 14647.604} C_VEL
LIN {X 0,Y 352.566,Z 1185.925,A -85,B 0,C 180,E1 14643.742,E2 14643.742} C_VEL
LIN {X 0,Y 356.582,Z 1174.584,A -85,B 0,C 180,E1 14640.429,E2 14640.429} C_VEL
LIN {X 0,Y 361.788,Z 1160.633,A -85,B 0,C 180,E1 14637.014,E2 14637.014} C_VEL
